C03632=1078.850,415.246,-107.346,176.673,31.266,155.541
C03633=1078.842,414.999,-107.303,176.669,31.256,155.538
C03634=1078.836,414.753,-107.261,176.663,31.246,155.536
C03635=1078.829,414.506,-107.218,176.659,31.236,155.534
C03636=1078.821,414.260,-107.176,176.654,31.226,155.532
C03637=1078.814,414.014,-107.134,176.649,31.216,155.530
C03638=1078.807,413.768,-107.091,176.645,31.206,155.528
C03639=1078.800,413.524,-107.050,176.640,31.197,155.526
C03640=1078.793,413.280,-107.008,176.635,31.187,155.523
C03641=1078.786,413.038,-106.966,176.630,31.177,155.521
C03642=1078.779,412.794,-106.924,176.626,31.167,155.519
C03643=1078.772,412.551,-106.883,176.622,31.158,155.517
C03644=1078.765,412.307,-106.841,176.617,31.148,155.515
C03645=1078.758,412.064,-106.799,176.612,31.139,155.513
C03646=1078.751,411.820,-106.757,176.607,31.129,155.511
C03647=1078.744,411.574,-106.716,176.603,31.119,155.509
C03648=1078.737,411.328,-106.674,176.599,31.110,155.507
C03649=1078.730,411.081,-106.631,176.593,31.100,155.505
C03650=1078.723,410.835,-106.590,176.589,31.091,155.503
C03651=1078.716,410.588,-106.547,176.584,31.081,155.501
C03652=1078.710,410.342,-106.506,176.580,31.072,155.499
C03653=1078.702,410.096,-106.464,176.576,31.062,155.496
C03654=1078.696,409.849,-106.422,176.570,31.053,155.494
C03655=1078.689,409.603,-106.380,176.566,31.043,155.492
C03656=1078.682,409.356,-106.338,176.562,31.034,155.490
C03657=1078.674,409.111,-106.296,176.557,31.024,155.488
C03658=1078.668,408.864,-106.255,176.553,31.015,155.486
C03659=1078.661,408.617,-106.213,176.548,31.006,155.484
C03660=1078.654,408.371,-106.171,176.543,30.996,155.482
C03661=1078.648,408.125,-106.129,176.539,30.987,155.480
C03662=1078.641,407.878,-106.088,176.534,30.977,155.478
C03663=1078.634,407.631,-106.046,176.530,30.968,155.476
C03664=1078.627,407.386,-106.005,176.526,30.959,155.474
C03665=1078.620,407.139,-105.963,176.521,30.950,155.472
C03666=1078.613,406.892,-105.922,176.517,30.941,155.470
C03667=1078.606,406.646,-105.880,176.513,30.932,155.469
C03668=1078.600,406.399,-105.839,176.508,30.922,155.466
C03669=1078.593,406.153,-105.798,176.504,30.913,155.465
C03670=1078.585,405.906,-105.757,176.500,30.904,155.463
C03671=1078.579,405.660,-105.715,176.494,30.895,155.461
C03672=1078.572,405.413,-105.674,176.490,30.886,155.459
C03673=1078.566,405.167,-105.632,176.485,30.877,155.457
C03674=1078.559,404.921,-105.591,176.481,30.869,155.455
C03675=1078.552,404.674,-105.550,176.477,30.860,155.453
C03676=1078.544,404.427,-105.509,176.472,30.851,155.451
C03677=1078.538,404.181,-105.467,176.468,30.841,155.449
C03678=1078.531,403.935,-105.426,176.464,30.833,155.448
C03679=1078.524,403.687,-105.386,176.459,30.824,155.446
C03680=1078.517,403.442,-105.345,176.455,30.815,155.444
C03681=1078.510,403.195,-105.303,176.451,30.806,155.442
C03682=1078.503,402.949,-105.263,176.446,30.798,155.440
C03683=1078.497,402.702,-105.221,176.442,30.789,155.438
C03684=1078.490,402.455,-105.180,176.438,30.780,155.436
C03685=1078.483,402.209,-105.139,176.433,30.772,155.435
C03686=1078.476,401.962,-105.099,176.429,30.763,155.433
C03687=1078.470,401.716,-105.058,176.425,30.755,155.431
C03688=1078.462,401.469,-105.017,176.421,30.746,155.429
C03689=1078.456,401.223,-104.977,176.417,30.738,155.427
C03690=1078.449,400.976,-104.935,176.413,30.729,155.426
C03691=1078.442,400.730,-104.895,176.408,30.721,155.424
C03692=1078.435,400.483,-104.854,176.404,30.712,155.422
C03693=1078.429,400.237,-104.814,176.400,30.703,155.420
C03694=1078.422,399.989,-104.773,176.395,30.695,155.418
C03695=1078.415,399.747,-104.733,176.391,30.686,155.417
C03696=1078.408,399.505,-104.693,176.387,30.678,155.415
C03697=1078.402,399.263,-104.653,176.383,30.670,155.413
C03698=1078.395,399.021,-104.613,176.379,30.662,155.411
C03699=1078.389,398.779,-104.574,176.375,30.653,155.410
C03700=1078.383,398.536,-104.535,176.370,30.645,155.408
C03701=1078.376,398.295,-104.495,176.366,30.637,155.406
C03702=1078.370,398.052,-104.455,176.363,30.629,155.405
C03703=1078.362,397.805,-104.415,176.358,30.621,155.403
C03704=1078.355,397.559,-104.374,176.354,30.613,155.401
C03705=1078.348,397.312,-104.333,176.350,30.604,155.400
C03706=1078.342,397.065,-104.293,176.345,30.596,155.398
C03707=1078.336,396.819,-104.253,176.342,30.588,155.396
C03708=1078.329,396.572,-104.213,176.338,30.580,155.394
C03709=1078.321,396.325,-104.173,176.333,30.572,155.393
C03710=1078.315,396.079,-104.133,176.329,30.564,155.391
C03711=1078.309,395.832,-104.093,176.325,30.555,155.389
C03712=1078.302,395.586,-104.053,176.320,30.547,155.388
C03713=1078.295,395.338,-104.012,176.317,30.539,155.386
C03714=1078.288,395.092,-103.973,176.313,30.531,155.384
C03715=1078.282,394.846,-103.932,176.309,30.523,155.383
C03716=1078.275,394.599,-103.892,176.304,30.515,155.381
C03717=1078.269,394.352,-103.852,176.301,30.507,155.379
C03718=1078.261,394.106,-103.812,176.297,30.499,155.378
C03719=1078.255,393.859,-103.773,176.292,30.491,155.376
C03720=1078.249,393.612,-103.733,176.288,30.484,155.375
C03721=1078.242,393.366,-103.693,176.284,30.476,155.373
C03722=1078.235,393.119,-103.653,176.280,30.468,155.371
C03723=1078.225,392.731,-103.591,176.273,30.455,155.369
C03724=1078.214,392.342,-103.528,176.268,30.443,155.366
C03725=1078.204,391.954,-103.466,176.261,30.430,155.364
C03726=1078.193,391.566,-103.403,176.255,30.418,155.361
C03727=1078.187,391.319,-103.363,176.250,30.411,155.360
C03728=1078.180,391.072,-103.324,176.246,30.403,155.358
C03729=1078.174,390.825,-103.284,176.243,30.396,155.356
C03730=1078.167,390.579,-103.245,176.238,30.388,155.355
C03731=1078.160,390.332,-103.206,176.234,30.380,155.353
C03732=1078.153,390.086,-103.166,176.230,30.372,155.352
C03733=1078.147,389.839,-103.127,176.227,30.365,155.350
C03734=1078.140,389.592,-103.087,176.222,30.357,155.349
C03735=1078.133,389.346,-103.048,176.218,30.350,155.347
C03736=1078.127,389.099,-103.009,176.215,30.343,155.346
C03737=1078.120,388.852,-102.969,176.210,30.335,155.344
C03738=1078.113,388.605,-102.930,176.206,30.327,155.343
C03739=1078.107,388.359,-102.891,176.203,30.320,155.341
C03740=1078.101,388.111,-102.852,176.198,30.312,155.340
C03741=1078.093,387.865,-102.812,176.194,30.305,155.338
C03742=1078.087,387.618,-102.774,176.191,30.298,155.337
C03743=1078.081,387.371,-102.734,176.187,30.290,155.335
C03744=1078.074,387.124,-102.695,176.182,30.283,155.334
C03745=1078.067,386.878,-102.657,176.179,30.276,155.332
C03746=1078.061,386.631,-102.616,176.175,30.268,155.331
C03747=1078.054,386.384,-102.578,176.170,30.261,155.329
C03748=1078.047,386.137,-102.539,176.167,30.253,155.328
C03749=1078.041,385.891,-102.500,176.163,30.246,155.326
C03750=1078.035,385.644,-102.461,176.159,30.239,155.325
C03751=1078.026,385.316,-102.409,176.153,30.229,155.323
C03752=1078.017,384.987,-102.357,176.148,30.219,155.321
C03753=1078.009,384.660,-102.306,176.143,30.210,155.319
C03754=1078.000,384.331,-102.254,176.138,30.200,155.317
C03755=1077.993,384.085,-102.215,176.135,30.193,155.316
C03756=1077.986,383.838,-102.176,176.131,30.186,155.314
C03757=1077.980,383.592,-102.138,176.126,30.179,155.313
C03758=1077.974,383.344,-102.099,176.123,30.171,155.311
C03759=1077.968,383.097,-102.060,176.119,30.164,155.310
C03760=1077.961,382.850,-102.021,176.115,30.157,155.308
C03761=1077.955,382.604,-101.983,176.111,30.150,155.307
C03762=1077.948,382.357,-101.945,176.108,30.143,155.306
C03763=1077.942,382.110,-101.905,176.104,30.136,155.304
C03764=1077.936,381.863,-101.867,176.099,30.129,155.303
C03765=1077.929,381.616,-101.829,176.096,30.122,155.301
C03766=1077.922,381.369,-101.790,176.092,30.114,155.300
C03767=1077.916,381.122,-101.751,176.088,30.108,155.299
C03768=1077.910,380.876,-101.713,176.084,30.101,155.297
C03769=1077.902,380.629,-101.675,176.081,30.094,155.296
C03770=1077.896,380.382,-101.637,176.077,30.087,155.294
C03771=1077.889,380.135,-101.598,176.073,30.080,155.293
C03772=1077.883,379.888,-101.560,176.069,30.073,155.292
C03773=1077.876,379.641,-101.521,176.066,30.066,155.290
C03774=1077.870,379.394,-101.483,176.061,30.059,155.289
C03775=1077.863,379.148,-101.445,176.058,30.052,155.288
C03776=1077.857,378.900,-101.407,176.054,30.046,155.286
C03777=1077.851,378.654,-101.368,176.050,30.039,155.285
C03778=1077.844,378.407,-101.330,176.046,30.032,155.284
C03779=1077.838,378.159,-101.292,176.043,30.025,155.282
C03780=1077.831,377.913,-101.254,176.039,30.018,155.281
C03781=1077.824,377.666,-101.216,176.035,30.012,155.280
C03782=1077.818,377.419,-101.178,176.031,30.005,155.278
C03783=1077.812,377.172,-101.140,176.028,29.998,155.277
C03784=1077.805,376.925,-101.101,176.023,29.991,155.276
C03785=1077.799,376.678,-101.064,176.020,29.985,155.274
C03786=1077.793,376.431,-101.025,176.016,29.978,155.273
C03787=1077.786,376.184,-100.988,176.013,29.971,155.272
C03788=1077.779,375.937,-100.950,176.009,29.965,155.270
C03789=1077.774,375.690,-100.912,176.005,29.958,155.269
C03790=1077.767,375.443,-100.874,176.002,29.951,155.268
C03791=1077.761,375.197,-100.836,175.997,29.944,155.266
C03792=1077.754,374.949,-100.798,175.994,29.938,155.265
C03793=1077.748,374.703,-100.760,175.990,29.931,155.264
C03794=1077.741,374.455,-100.722,175.987,29.925,155.263
C03795=1077.735,374.209,-100.685,175.983,29.918,155.261
C03796=1077.729,373.961,-100.646,175.979,29.911,155.260
C03797=1077.723,373.714,-100.609,175.976,29.905,155.259
C03798=1077.716,373.468,-100.572,175.971,29.898,155.257
C03799=1077.710,373.220,-100.533,175.968,29.892,155.256
C03800=1077.703,372.973,-100.497,175.965,29.886,155.255
C03801=1077.697,372.726,-100.459,175.960,29.879,155.254
C03802=1077.691,372.479,-100.421,175.957,29.872,155.252
C03803=1077.685,372.258,-100.388,175.954,29.867,155.251
C03804=1077.679,372.038,-100.354,175.950,29.861,155.250
C03805=1077.673,371.818,-100.321,175.947,29.855,155.249
C03806=1077.668,371.597,-100.287,175.944,29.849,155.248
C03807=1077.661,371.377,-100.254,175.940,29.844,155.247
C03808=1077.656,371.156,-100.221,175.937,29.838,155.246
C03809=1077.651,370.935,-100.187,175.934,29.832,155.245
C03810=1077.645,370.714,-100.154,175.931,29.827,155.244
C03811=1077.638,370.468,-100.117,175.927,29.820,155.242
C03812=1077.632,370.221,-100.079,175.924,29.814,155.241
C03813=1077.625,369.973,-100.042,175.919,29.808,155.240
C03814=1077.619,369.727,-100.004,175.916,29.802,155.239
C03815=1077.612,369.479,-99.968,175.913,29.795,155.238
C03816=1077.606,369.232,-99.930,175.908,29.789,155.236
C03817=1077.600,368.986,-99.893,175.905,29.782,155.235
C03818=1077.594,368.738,-99.856,175.902,29.776,155.234
C03819=1077.587,368.491,-99.818,175.898,29.770,155.233
C03820=1077.581,368.244,-99.781,175.894,29.764,155.232
C03821=1077.575,367.997,-99.745,175.891,29.758,155.230
C03822=1077.568,367.749,-99.706,175.887,29.751,155.229
C03823=1077.562,367.502,-99.670,175.883,29.745,155.228
C03824=1077.555,367.256,-99.633,175.880,29.739,155.227
C03825=1077.550,367.008,-99.596,175.877,29.733,155.226
C03826=1077.543,366.761,-99.559,175.873,29.726,155.224
C03827=1077.537,366.514,-99.521,175.869,29.720,155.223
C03828=1077.531,366.267,-99.485,175.866,29.714,155.222
C03829=1077.525,366.020,-99.448,175.862,29.708,155.221
C03830=1077.518,365.773,-99.411,175.858,29.702,155.220
C03831=1077.512,365.525,-99.374,175.855,29.696,155.219
C03832=1077.506,365.278,-99.337,175.851,29.689,155.217
C03833=1077.500,365.031,-99.300,175.848,29.683,155.216
C03834=1077.493,364.784,-99.264,175.844,29.677,155.215
C03835=1077.487,364.537,-99.226,175.841,29.671,155.214
C03836=1077.480,364.289,-99.189,175.837,29.666,155.213
C03837=1077.474,364.042,-99.153,175.833,29.659,155.212
C03838=1077.468,363.795,-99.116,175.830,29.653,155.211
C03839=1077.461,363.548,-99.080,175.827,29.647,155.209
C03840=1077.456,363.301,-99.043,175.822,29.641,155.208
C03841=1077.449,363.053,-99.006,175.819,29.636,155.207
C03842=1077.443,362.806,-98.970,175.816,29.630,155.206
C03843=1077.436,362.559,-98.933,175.813,29.624,155.205
C03844=1077.430,362.312,-98.897,175.808,29.617,155.204
C03845=1077.423,362.065,-98.860,175.805,29.612,155.203
C03846=1077.417,361.818,-98.824,175.802,29.606,155.202
C03847=1077.412,361.570,-98.787,175.798,29.600,155.201
C03848=1077.405,361.323,-98.750,175.794,29.594,155.199
C03849=1077.398,361.076,-98.714,175.791,29.588,155.198
C03850=1077.392,360.828,-98.678,175.787,29.582,155.197
C03851=1077.386,360.581,-98.641,175.784,29.576,155.196
C03852=1077.380,360.334,-98.605,175.781,29.571,155.195
C03853=1077.373,360.087,-98.569,175.777,29.564,155.194
C03854=1077.367,359.840,-98.532,175.773,29.559,155.193
C03855=1077.361,359.592,-98.496,175.770,29.553,155.192
C03856=1077.355,359.345,-98.460,175.767,29.547,155.191
C03857=1077.348,359.098,-98.423,175.763,29.541,155.190
C03858=1077.342,358.851,-98.387,175.759,29.535,155.188
C03859=1077.337,358.638,-98.356,175.757,29.531,155.188
C03860=1077.331,358.426,-98.325,175.753,29.526,155.187
C03861=1077.326,358.213,-98.294,175.750,29.521,155.186
C03862=1077.320,358.001,-98.263,175.747,29.516,155.185
C03863=1077.315,357.789,-98.232,175.744,29.511,155.184
C03864=1077.309,357.576,-98.201,175.742,29.506,155.183
C03865=1077.305,357.364,-98.170,175.738,29.501,155.182
C03866=1077.299,357.152,-98.139,175.736,29.496,155.181
C03867=1077.293,356.905,-98.103,175.732,29.490,155.180
C03868=1077.287,356.657,-98.067,175.728,29.485,155.179
C03869=1077.280,356.410,-98.031,175.725,29.479,155.178
C03870=1077.274,356.162,-97.995,175.722,29.474,155.177
C03871=1077.268,355.915,-97.959,175.718,29.468,155.176
C03872=1077.262,355.667,-97.923,175.715,29.462,155.175
C03873=1077.255,355.420,-97.887,175.711,29.456,155.174
C03874=1077.249,355.173,-97.851,175.707,29.451,155.173
C03875=1077.243,354.925,-97.816,175.704,29.445,155.172
C03876=1077.236,354.678,-97.779,175.701,29.439,155.171
C03877=1077.231,354.431,-97.744,175.698,29.434,155.170
C03878=1077.225,354.184,-97.708,175.694,29.428,155.169
C03879=1077.219,353.937,-97.672,175.691,29.423,155.168
C03880=1077.212,353.689,-97.636,175.688,29.417,155.167
C03881=1077.206,353.442,-97.601,175.683,29.411,155.166
C03882=1077.200,353.194,-97.565,175.680,29.406,155.165
C03883=1077.193,352.947,-97.529,175.677,29.400,155.164
C03884=1077.188,352.700,-97.493,175.673,29.395,155.163
C03885=1077.181,352.452,-97.458,175.670,29.390,155.162
C03886=1077.175,352.205,-97.422,175.667,29.384,155.161
C03887=1077.169,351.957,-97.387,175.664,29.378,155.160
C03888=1077.162,351.710,-97.352,175.660,29.373,155.159
C03889=1077.156,351.463,-97.315,175.657,29.368,155.158
C03890=1077.150,351.215,-97.279,175.653,29.362,155.157
C03891=1077.144,350.968,-97.245,175.649,29.356,155.156
C03892=1077.138,350.721,-97.209,175.646,29.351,155.155
C03893=1077.132,350.473,-97.173,175.643,29.346,155.154
C03894=1077.125,350.226,-97.138,175.639,29.340,155.153
C03895=1077.119,349.978,-97.102,175.636,29.335,155.152
C03896=1077.113,349.731,-97.068,175.633,29.330,155.151
C03897=1077.107,349.484,-97.032,175.629,29.324,155.150
C03898=1077.100,349.236,-96.997,175.626,29.319,155.149
C03899=1077.094,348.988,-96.962,175.623,29.313,155.148
C03900=1077.089,348.741,-96.926,175.620,29.308,155.147
C03901=1077.082,348.494,-96.891,175.616,29.303,155.146
C03902=1077.076,348.246,-96.855,175.613,29.297,155.145
C03903=1077.069,347.999,-96.820,175.610,29.292,155.144
C03904=1077.064,347.752,-96.785,175.605,29.286,155.143
C03905=1077.057,347.504,-96.750,175.602,29.281,155.142
C03906=1077.051,347.256,-96.715,175.599,29.275,155.141
C03907=1077.045,347.009,-96.680,175.595,29.270,155.140
C03908=1077.039,346.762,-96.644,175.592,29.265,155.139
C03909=1077.033,346.514,-96.610,175.589,29.260,155.138
C03910=1077.027,346.267,-96.574,175.585,29.255,155.137
C03911=1077.020,346.019,-96.539,175.582,29.249,155.136
C03912=1077.014,345.772,-96.504,175.579,29.244,155.135
C03913=1077.009,345.524,-96.470,175.576,29.239,155.134
C03914=1077.003,345.277,-96.434,175.572,29.233,155.133
C03915=1076.997,345.066,-96.404,175.570,29.229,155.133
C03916=1076.992,344.855,-96.375,175.566,29.224,155.132
C03917=1076.987,344.645,-96.345,175.564,29.220,155.131
C03918=1076.982,344.434,-96.316,175.562,29.216,155.130
C03919=1076.977,344.223,-96.285,175.558,29.211,155.129
C03920=1076.971,344.013,-96.255,175.556,29.207,155.129
C03921=1076.966,343.802,-96.226,175.552,29.202,155.128
C03922=1076.960,343.591,-96.197,175.550,29.198,155.127
C03923=1076.955,343.343,-96.162,175.547,29.193,155.126
C03924=1076.948,343.096,-96.127,175.543,29.188,155.125
C03925=1076.942,342.848,-96.092,175.540,29.183,155.124
C03926=1076.935,342.601,-96.057,175.537,29.177,155.123
C03927=1076.930,342.353,-96.023,175.533,29.172,155.122
C03928=1076.924,342.105,-95.988,175.530,29.167,155.121
C03929=1076.917,341.859,-95.954,175.527,29.162,155.121
C03930=1076.911,341.611,-95.919,175.523,29.156,155.120
C03931=1076.906,341.363,-95.884,175.520,29.151,155.119
C03932=1076.899,341.116,-95.849,175.517,29.146,155.118
C03933=1076.893,340.868,-95.815,175.514,29.141,155.117
C03934=1076.887,340.620,-95.781,175.510,29.136,155.116
C03935=1076.881,340.374,-95.746,175.507,29.131,155.115
C03936=1076.875,340.125,-95.711,175.504,29.126,155.114
C03937=1076.869,339.878,-95.677,175.500,29.121,155.113
C03938=1076.862,339.630,-95.643,175.497,29.116,155.112
C03939=1076.856,339.383,-95.608,175.494,29.111,155.112
C03940=1076.850,339.135,-95.573,175.491,29.106,155.111
C03941=1076.844,338.888,-95.539,175.488,29.101,155.110
C03942=1076.838,338.640,-95.504,175.485,29.095,155.109
C03943=1076.832,338.393,-95.470,175.481,29.091,155.108
C03944=1076.826,338.145,-95.436,175.478,29.086,155.107
C03945=1076.820,337.897,-95.402,175.475,29.081,155.106
C03946=1076.814,337.649,-95.367,175.471,29.076,155.105
C03947=1076.808,337.402,-95.333,175.468,29.070,155.104
C03948=1076.801,337.154,-95.299,175.465,29.066,155.104
C03949=1076.795,336.907,-95.265,175.461,29.061,155.103
C03950=1076.790,336.660,-95.231,175.458,29.056,155.102
C03951=1076.783,336.412,-95.196,175.455,29.050,155.101
C03952=1076.777,336.164,-95.162,175.452,29.046,155.100
C03953=1076.771,335.916,-95.128,175.449,29.041,155.099
C03954=1076.765,335.669,-95.094,175.446,29.036,155.098
C03955=1076.758,335.421,-95.059,175.443,29.031,155.098
C03956=1076.753,335.174,-95.025,175.439,29.026,155.097
C03957=1076.747,334.926,-94.991,175.436,29.021,155.096
C03958=1076.740,334.678,-94.957,175.433,29.016,155.095
C03959=1076.735,334.431,-94.924,175.429,29.011,155.094
C03960=1076.729,334.183,-94.890,175.426,29.006,155.093
C03961=1076.722,333.936,-94.856,175.424,29.002,155.092
C03962=1076.716,333.688,-94.822,175.420,28.997,155.092
C03963=1076.710,333.441,-94.788,175.417,28.992,155.091
C03964=1076.704,333.192,-94.754,175.414,28.987,155.090
C03965=1076.698,332.945,-94.720,175.410,28.982,155.089
C03966=1076.692,332.698,-94.686,175.407,28.977,155.088
C03967=1076.686,332.449,-94.652,175.404,28.972,155.087
C03968=1076.680,332.202,-94.618,175.400,28.967,155.087
C03969=1076.674,331.955,-94.584,175.398,28.962,155.086
C03970=1076.669,331.707,-94.551,175.395,28.958,155.085
C03971=1076.662,331.494,-94.522,175.391,28.953,155.084
C03972=1076.657,331.280,-94.492,175.389,28.949,155.083
C03973=1076.653,331.067,-94.463,175.387,28.946,155.083
C03974=1076.647,330.853,-94.435,175.384,28.941,155.082
C03975=1076.641,330.640,-94.405,175.381,28.937,155.081
C03976=1076.636,330.426,-94.376,175.378,28.933,155.081
C03977=1076.631,330.214,-94.348,175.376,28.929,155.080
C03978=1076.625,330.000,-94.319,175.372,28.925,155.079
C03979=1076.620,329.752,-94.285,175.369,28.920,155.078
C03980=1076.613,329.504,-94.252,175.367,28.916,155.078
C03981=1076.607,329.257,-94.218,175.363,28.911,155.077
C03982=1076.600,329.009,-94.185,175.360,28.906,155.076
C03983=1076.595,328.761,-94.151,175.357,28.901,155.075
C03984=1076.588,328.514,-94.118,175.353,28.897,155.074
C03985=1076.582,328.266,-94.084,175.351,28.892,155.074
C03986=1076.576,328.019,-94.051,175.348,28.888,155.073
C03987=1076.570,327.771,-94.017,175.344,28.883,155.072
C03988=1076.563,327.523,-93.984,175.341,28.878,155.071
C03989=1076.557,327.275,-93.950,175.338,28.873,155.070
C03990=1076.551,327.028,-93.918,175.334,28.869,155.070
C03991=1076.545,326.780,-93.884,175.332,28.864,155.069
C03992=1076.539,326.532,-93.851,175.329,28.860,155.068
C03993=1076.533,326.284,-93.817,175.325,28.854,155.067
C03994=1076.527,326.036,-93.784,175.322,28.850,155.066
C03995=1076.521,325.789,-93.751,175.320,28.845,155.066
C03996=1076.515,325.541,-93.718,175.316,28.841,155.065
C03997=1076.509,325.294,-93.684,175.313,28.836,155.064
C03998=1076.502,325.046,-93.651,175.310,28.832,155.063
C03999=1076.497,324.798,-93.618,175.306,28.827,155.063
C04000=1076.490,324.550,-93.585,175.304,28.822,155.062
C04001=1076.484,324.302,-93.552,175.301,28.818,155.061
C04002=1076.478,324.054,-93.519,175.298,28.813,155.060
C04003=1076.473,323.807,-93.486,175.294,28.808,155.059
C04004=1076.466,323.559,-93.453,175.292,28.804,155.059
C04005=1076.460,323.312,-93.419,175.289,28.799,155.058
C04006=1076.454,323.064,-93.386,175.285,28.794,155.057
C04007=1076.449,322.816,-93.353,175.282,28.790,155.056
C04008=1076.442,322.569,-93.320,175.280,28.785,155.055
C04009=1076.436,322.321,-93.287,175.276,28.781,155.055
C04010=1076.430,322.073,-93.254,175.273,28.776,155.054
C04011=1076.424,321.826,-93.221,175.270,28.771,155.053
C04012=1076.419,321.577,-93.189,175.267,28.767,155.052
C04013=1076.413,321.329,-93.156,175.264,28.762,155.052
C04014=1076.406,321.082,-93.123,175.261,28.758,155.051
C04015=1076.401,320.834,-93.090,175.258,28.753,155.050
C04016=1076.394,320.586,-93.057,175.255,28.749,155.049
C04017=1076.389,320.338,-93.024,175.252,28.744,155.048
C04018=1076.383,320.091,-92.991,175.248,28.739,155.048
C04019=1076.376,319.843,-92.958,175.246,28.735,155.047
C04020=1076.371,319.595,-92.925,175.243,28.730,155.046
C04021=1076.365,319.347,-92.893,175.239,28.726,155.045
C04022=1076.358,319.100,-92.860,175.237,28.721,155.045
C04023=1076.353,318.852,-92.827,175.234,28.717,155.044
C04024=1076.347,318.604,-92.794,175.230,28.712,155.043
C04025=1076.341,318.357,-92.762,175.227,28.708,155.042
C04026=1076.336,318.109,-92.729,175.225,28.703,155.042
C04027=1076.330,317.892,-92.701,175.222,28.699,155.041
C04028=1076.325,317.675,-92.672,175.219,28.695,155.040
C04029=1076.321,317.459,-92.643,175.216,28.691,155.040
C04030=1076.315,317.242,-92.615,175.214,28.687,155.039
C04031=1076.310,317.026,-92.586,175.212,28.683,155.038
C04032=1076.304,316.809,-92.557,175.208,28.679,155.038
C04033=1076.300,316.593,-92.529,175.206,28.675,155.037
C04034=1076.294,316.376,-92.501,175.203,28.671,155.036
C04035=1076.289,316.127,-92.468,175.200,28.666,155.035
C04036=1076.282,315.880,-92.435,175.198,28.663,155.035
C04037=1076.277,315.632,-92.404,175.194,28.658,155.034
C04038=1076.271,315.384,-92.370,175.191,28.653,155.033
C04039=1076.265,315.137,-92.337,175.189,28.649,155.032
C04040=1076.259,314.889,-92.305,175.185,28.644,155.032
C04041=1076.253,314.642,-92.273,175.182,28.640,155.031
C04042=1076.247,314.393,-92.241,175.180,28.636,155.030
C04043=1076.241,314.145,-92.209,175.176,28.631,155.030
C04044=1076.235,313.898,-92.176,175.173,28.627,155.029
C04045=1076.229,313.649,-92.144,175.171,28.622,155.028
C04046=1076.223,313.402,-92.112,175.167,28.618,155.027
C04047=1076.217,313.154,-92.079,175.164,28.614,155.027
C04048=1076.210,312.906,-92.048,175.162,28.610,155.026
C04049=1076.204,312.659,-92.016,175.158,28.605,155.025
C04050=1076.198,312.411,-91.984,175.155,28.601,155.025
C04051=1076.192,312.162,-91.952,175.153,28.596,155.024
C04052=1076.186,311.915,-91.919,175.149,28.592,155.023
C04053=1076.180,311.667,-91.887,175.146,28.588,155.022
C04054=1076.174,311.419,-91.856,175.144,28.584,155.022
C04055=1076.168,311.172,-91.823,175.140,28.579,155.021
C04056=1076.162,310.924,-91.791,175.138,28.575,155.020
C04057=1076.156,310.675,-91.759,175.135,28.570,155.020
C04058=1076.150,310.428,-91.727,175.131,28.566,155.019
C04059=1076.144,310.180,-91.696,175.129,28.562,155.018
C04060=1076.137,309.932,-91.663,175.126,28.558,155.017
C04061=1076.131,309.684,-91.631,175.122,28.553,155.017
C04062=1076.126,309.437,-91.599,175.120,28.549,155.016
C04063=1076.120,309.188,-91.567,175.117,28.544,155.015
C04064=1076.113,308.941,-91.536,175.113,28.540,155.015
C04065=1076.107,308.692,-91.504,175.111,28.536,155.014
C04066=1076.102,308.445,-91.472,175.108,28.532,155.013
C04067=1076.096,308.197,-91.440,175.105,28.528,155.013
C04068=1076.089,307.949,-91.408,175.102,28.523,155.012
C04069=1076.084,307.702,-91.376,175.099,28.519,155.011
C04070=1076.078,307.454,-91.344,175.096,28.514,155.010
C04071=1076.072,307.206,-91.313,175.093,28.510,155.010
C04072=1076.065,306.958,-91.281,175.091,28.506,155.009
C04073=1076.059,306.710,-91.249,175.087,28.502,155.008
C04074=1076.054,306.462,-91.218,175.084,28.497,155.008
C04075=1076.047,306.215,-91.186,175.082,28.493,155.007
C04076=1076.041,305.966,-91.154,175.078,28.489,155.006
C04077=1076.036,305.719,-91.123,175.076,28.485,155.006
C04078=1076.030,305.471,-91.091,175.073,28.480,155.005
C04079=1076.024,305.223,-91.060,175.069,28.476,155.004
C04080=1076.018,304.975,-91.028,175.067,28.472,155.003
C04081=1076.013,304.727,-90.996,175.064,28.467,155.003
C04082=1076.006,304.479,-90.965,175.061,28.463,155.002
C04083=1076.002,304.264,-90.938,175.059,28.460,155.001
C04084=1075.996,304.049,-90.911,175.055,28.456,155.001
C04085=1075.992,303.834,-90.882,175.053,28.452,155.000
C04086=1075.986,303.619,-90.855,175.051,28.449,155.000
C04087=1075.980,303.404,-90.828,175.048,28.445,154.999
C04088=1075.976,303.189,-90.801,175.046,28.441,154.998
C04089=1075.971,302.974,-90.774,175.043,28.437,154.998
C04090=1075.965,302.759,-90.746,175.041,28.433,154.997
C04091=1075.960,302.511,-90.715,175.038,28.429,154.997
C04092=1075.954,302.263,-90.683,175.035,28.425,154.996
C04093=1075.948,302.016,-90.652,175.032,28.421,154.995
C04094=1075.942,301.767,-90.620,175.030,28.417,154.994
C04095=1075.936,301.520,-90.590,175.026,28.412,154.994
C04096=1075.931,301.272,-90.558,175.024,28.408,154.993
C04097=1075.925,301.024,-90.526,175.021,28.404,154.992
C04098=1075.919,300.776,-90.496,175.018,28.400,154.992
C04099=1075.913,300.528,-90.464,175.015,28.395,154.991
C04100=1075.908,300.280,-90.433,175.012,28.391,154.990
C04101=1075.901,300.032,-90.401,175.009,28.387,154.990
C04102=1075.896,299.784,-90.370,175.006,28.382,154.989
C04103=1075.890,299.537,-90.339,175.004,28.378,154.988
C04104=1075.884,299.288,-90.307,175.000,28.374,154.988
C04105=1075.878,299.041,-90.277,174.998,28.370,154.987
C04106=1075.873,298.793,-90.245,174.995,28.366,154.986
C04107=1075.867,298.544,-90.214,174.992,28.362,154.986
C04108=1075.861,298.297,-90.183,174.989,28.357,154.985
C04109=1075.856,298.049,-90.152,174.987,28.353,154.984
C04110=1075.849,297.801,-90.120,174.983,28.349,154.984
C04111=1075.844,297.553,-90.090,174.981,28.345,154.983
C04112=1075.838,297.304,-90.059,174.978,28.340,154.982
C04113=1075.832,297.057,-90.028,174.975,28.336,154.981
C04114=1075.826,296.809,-89.997,174.972,28.332,154.981
C04115=1075.820,296.560,-89.966,174.970,28.328,154.980
C04116=1075.814,296.313,-89.935,174.966,28.324,154.980
C04117=1075.808,296.064,-89.904,174.964,28.320,154.979
C04118=1075.802,295.817,-89.873,174.961,28.316,154.978
C04119=1075.796,295.569,-89.842,174.958,28.311,154.977
C04120=1075.791,295.321,-89.811,174.955,28.307,154.977
C04121=1075.785,295.073,-89.781,174.953,28.303,154.976
C04122=1075.779,294.825,-89.750,174.949,28.299,154.976
C04123=1075.772,294.577,-89.719,174.947,28.295,154.975
C04124=1075.766,294.329,-89.688,174.944,28.291,154.974
C04125=1075.761,294.081,-89.658,174.941,28.287,154.974
C04126=1075.755,293.833,-89.627,174.938,28.283,154.973
C04127=1075.749,293.585,-89.596,174.936,28.279,154.972
C04128=1075.743,293.337,-89.565,174.932,28.274,154.972
C04129=1075.737,293.089,-89.535,174.930,28.270,154.971
C04130=1075.731,292.841,-89.504,174.927,28.266,154.970
C04131=1075.726,292.593,-89.473,174.924,28.262,154.970
C04132=1075.720,292.345,-89.443,174.921,28.258,154.969
C04133=1075.713,292.097,-89.412,174.919,28.254,154.968
C04134=1075.708,291.849,-89.382,174.916,28.250,154.968
C04135=1075.702,291.601,-89.352,174.913,28.246,154.967
C04136=1075.696,291.352,-89.320,174.910,28.242,154.966
C04137=1075.690,291.104,-89.290,174.907,28.238,154.966
C04138=1075.684,290.857,-89.260,174.905,28.234,154.965
C04139=1075.675,290.441,-89.209,174.900,28.227,154.964
C04140=1075.664,290.026,-89.157,174.895,28.220,154.963
C04141=1075.655,289.610,-89.106,174.890,28.213,154.962
C04142=1075.645,289.195,-89.056,174.886,28.206,154.961
C04143=1075.640,288.947,-89.026,174.883,28.202,154.960
C04144=1075.633,288.698,-88.995,174.881,28.199,154.960
C04145=1075.627,288.450,-88.964,174.877,28.194,154.959
C04146=1075.621,288.203,-88.934,174.875,28.190,154.958
C04147=1075.615,287.955,-88.904,174.873,28.186,154.958
C04148=1075.609,287.706,-88.874,174.869,28.182,154.957
C04149=1075.603,287.458,-88.844,174.867,28.178,154.956
C04150=1075.597,287.210,-88.814,174.864,28.174,154.956
C04151=1075.591,286.963,-88.783,174.861,28.170,154.955
C04152=1075.586,286.714,-88.754,174.858,28.166,154.955
C04153=1075.579,286.466,-88.723,174.856,28.162,154.954
C04154=1075.574,286.218,-88.693,174.853,28.158,154.953
C04155=1075.568,285.970,-88.662,174.850,28.154,154.953
C04156=1075.562,285.722,-88.633,174.848,28.150,154.952
C04157=1075.556,285.474,-88.603,174.844,28.146,154.951
C04158=1075.550,285.226,-88.572,174.842,28.142,154.951
C04159=1075.544,284.978,-88.543,174.840,28.138,154.950
C04160=1075.538,284.729,-88.512,174.836,28.134,154.949
C04161=1075.532,284.481,-88.482,174.834,28.130,154.949
C04162=1075.527,284.233,-88.452,174.831,28.126,154.948
C04163=1075.521,283.985,-88.422,174.828,28.122,154.948
C04164=1075.515,283.737,-88.393,174.826,28.118,154.947
C04165=1075.509,283.489,-88.362,174.823,28.114,154.946
C04166=1075.503,283.241,-88.333,174.820,28.110,154.946
C04167=1075.497,282.993,-88.302,174.817,28.106,154.945
C04168=1075.492,282.744,-88.273,174.815,28.102,154.944
C04169=1075.486,282.497,-88.242,174.812,28.098,154.944
C04170=1075.480,282.249,-88.213,174.809,28.094,154.943
C04171=1075.474,282.001,-88.183,174.807,28.090,154.942
C04172=1075.469,281.752,-88.153,174.804,28.086,154.942
C04173=1075.463,281.504,-88.123,174.801,28.082,154.941
C04174=1075.457,281.256,-88.093,174.799,28.078,154.941
C04175=1075.451,281.007,-88.063,174.795,28.074,154.940
C04176=1075.445,280.759,-88.034,174.793,28.070,154.939
C04177=1075.439,280.511,-88.004,174.791,28.066,154.939
C04178=1075.433,280.263,-87.974,174.787,28.062,154.938
C04179=1075.427,280.015,-87.945,174.785,28.058,154.937
C04180=1075.421,279.766,-87.915,174.783,28.054,154.937
C04181=1075.415,279.519,-87.885,174.779,28.050,154.936
C04182=1075.409,279.271,-87.856,174.777,28.046,154.936
C04183=1075.404,279.022,-87.826,174.775,28.042,154.935
C04184=1075.398,278.774,-87.797,174.771,28.038,154.934
C04185=1075.392,278.526,-87.767,174.769,28.034,154.934
C04186=1075.386,278.278,-87.737,174.766,28.031,154.933
C04187=1075.380,278.030,-87.708,174.763,28.027,154.933
C04188=1075.375,277.781,-87.678,174.761,28.023,154.932
C04189=1075.368,277.534,-87.649,174.758,28.018,154.931
C04190=1075.362,277.285,-87.619,174.755,28.015,154.931
C04191=1075.353,276.880,-87.570,174.751,28.008,154.930
C04192=1075.343,276.474,-87.523,174.746,28.002,154.929
C04193=1075.334,276.069,-87.474,174.743,27.995,154.928
C04194=1075.325,275.664,-87.427,174.738,27.989,154.927
C04195=1075.319,275.416,-87.397,174.735,27.985,154.926
C04196=1075.313,275.168,-87.368,174.733,27.981,154.925
C04197=1075.307,274.919,-87.338,174.730,27.977,154.925
C04198=1075.301,274.671,-87.309,174.727,27.973,154.924
C04199=1075.295,274.423,-87.280,174.725,27.969,154.924
C04200=1075.289,274.174,-87.251,174.722,27.965,154.923
C04201=1075.284,273.926,-87.221,174.719,27.961,154.922
C04202=1075.277,273.678,-87.192,174.717,27.957,154.922
C04203=1075.272,273.429,-87.162,174.715,27.953,154.921
C04204=1075.266,273.182,-87.134,174.711,27.950,154.921
C04205=1075.260,272.933,-87.105,174.709,27.946,154.920
C04206=1075.255,272.685,-87.076,174.707,27.942,154.919
C04207=1075.249,272.437,-87.047,174.703,27.938,154.919
C04208=1075.242,272.189,-87.018,174.701,27.934,154.918
C04209=1075.237,271.940,-86.988,174.699,27.930,154.917
C04210=1075.230,271.692,-86.959,174.695,27.926,154.917
C04211=1075.224,271.444,-86.930,174.693,27.922,154.916
C04212=1075.219,271.196,-86.901,174.691,27.918,154.916
C04213=1075.213,270.947,-86.872,174.688,27.915,154.915
C04214=1075.207,270.699,-86.843,174.685,27.911,154.915
C04215=1075.202,270.451,-86.814,174.683,27.907,154.914
C04216=1075.195,270.203,-86.785,174.680,27.903,154.913
C04217=1075.189,269.954,-86.756,174.677,27.899,154.913
C04218=1075.185,269.706,-86.727,174.675,27.895,154.912
C04219=1075.178,269.458,-86.698,174.672,27.891,154.912
C04220=1075.172,269.210,-86.669,174.670,27.887,154.911
C04221=1075.166,268.961,-86.641,174.667,27.883,154.910
C04222=1075.161,268.713,-86.611,174.664,27.880,154.910
C04223=1075.155,268.465,-86.582,174.662,27.876,154.909
C04224=1075.149,268.216,-86.554,174.659,27.871,154.908
C04225=1075.143,267.968,-86.525,174.656,27.868,154.908
C04226=1075.136,267.720,-86.496,174.654,27.864,154.907
C04227=1075.132,267.472,-86.467,174.652,27.860,154.907
C04228=1075.126,267.224,-86.438,174.648,27.856,154.906
C04229=1075.120,266.975,-86.410,174.646,27.852,154.905
C04230=1075.113,266.727,-86.381,174.644,27.849,154.905
C04231=1075.108,266.479,-86.352,174.641,27.845,154.904
C04232=1075.102,266.231,-86.324,174.638,27.840,154.904
C04233=1075.096,265.982,-86.294,174.636,27.837,154.903
C04234=1075.090,265.733,-86.266,174.634,27.833,154.902
C04235=1075.085,265.486,-86.237,174.631,27.829,154.902
C04236=1075.079,265.237,-86.209,174.628,27.825,154.901
C04237=1075.073,264.989,-86.180,174.626,27.821,154.901
C04238=1075.067,264.741,-86.152,174.623,27.818,154.900
C04239=1075.061,264.492,-86.124,174.621,27.814,154.900
C04240=1075.055,264.244,-86.095,174.618,27.809,154.899
C04241=1075.050,263.995,-86.066,174.615,27.806,154.898
C04242=1075.044,263.748,-86.037,174.613,27.802,154.898
C04243=1075.034,263.345,-85.992,174.609,27.796,154.897
C04244=1075.024,262.943,-85.945,174.604,27.789,154.896
C04245=1075.015,262.541,-85.900,174.600,27.784,154.895
C04246=1075.005,262.139,-85.853,174.596,27.778,154.894
C04247=1074.999,261.890,-85.825,174.594,27.774,154.893
C04248=1074.993,261.641,-85.797,174.592,27.770,154.893
C04249=1074.987,261.393,-85.769,174.588,27.766,154.892
C04250=1074.981,261.145,-85.740,174.586,27.762,154.892
C04251=1074.975,260.897,-85.712,174.584,27.758,154.891
C04252=1074.969,260.649,-85.684,174.581,27.755,154.891
C04253=1074.963,260.400,-85.656,174.578,27.750,154.890
C04254=1074.957,260.151,-85.627,174.576,27.747,154.889
C04255=1074.952,259.904,-85.599,174.573,27.743,154.889
C04256=1074.946,259.655,-85.570,174.571,27.740,154.888
C04257=1074.939,259.407,-85.543,174.569,27.735,154.888
C04258=1074.934,259.159,-85.515,174.565,27.732,154.887
C04259=1074.928,258.910,-85.486,174.563,27.728,154.886
C04260=1074.922,258.661,-85.458,174.561,27.724,154.886
C04261=1074.916,258.413,-85.431,174.558,27.720,154.885
C04262=1074.910,258.165,-85.402,174.556,27.717,154.885
C04263=1074.904,257.917,-85.374,174.553,27.712,154.884
C04264=1074.898,257.668,-85.345,174.550,27.709,154.884
C04265=1074.892,257.420,-85.317,174.548,27.705,154.883
C04266=1074.886,257.172,-85.290,174.546,27.701,154.882
C04267=1074.880,256.923,-85.261,174.543,27.697,154.882
C04268=1074.875,256.675,-85.233,174.540,27.694,154.881
C04269=1074.869,256.426,-85.205,174.538,27.690,154.881
C04270=1074.863,256.179,-85.178,174.535,27.686,154.880
C04271=1074.857,255.930,-85.149,174.533,27.682,154.879
C04272=1074.852,255.682,-85.122,174.531,27.679,154.879
C04273=1074.846,255.432,-85.094,174.529,27.675,154.878
C04274=1074.839,255.184,-85.066,174.525,27.670,154.878
C04275=1074.834,254.936,-85.038,174.523,27.667,154.877
C04276=1074.828,254.687,-85.010,174.521,27.663,154.876
C04277=1074.822,254.439,-84.983,174.518,27.659,154.876
C04278=1074.816,254.191,-84.954,174.516,27.655,154.875
C04279=1074.811,253.943,-84.926,174.514,27.652,154.875
C04280=1074.805,253.695,-84.898,174.510,27.647,154.874
C04281=1074.799,253.446,-84.871,174.508,27.644,154.874
C04282=1074.794,253.198,-84.843,174.506,27.640,154.873
C04283=1074.788,252.949,-84.815,174.503,27.636,154.872
C04284=1074.782,252.701,-84.788,174.501,27.632,154.872
C04285=1074.776,252.452,-84.759,174.499,27.628,154.871
C04286=1074.771,252.204,-84.732,174.496,27.625,154.871
C04287=1074.764,251.955,-84.704,174.493,27.621,154.870
C04288=1074.759,251.707,-84.676,174.491,27.617,154.869
C04289=1074.753,251.459,-84.648,174.489,27.613,154.869
C04290=1074.747,251.210,-84.621,174.486,27.609,154.868
C04291=1074.741,250.962,-84.593,174.484,27.605,154.868
C04292=1074.736,250.713,-84.565,174.482,27.601,154.867
C04293=1074.730,250.465,-84.538,174.478,27.598,154.867
C04294=1074.724,250.217,-84.511,174.476,27.594,154.866
C04295=1074.715,249.811,-84.465,174.472,27.587,154.865
C04296=1074.705,249.407,-84.421,174.468,27.581,154.864
C04297=1074.696,249.002,-84.376,174.464,27.575,154.863
C04298=1074.687,248.597,-84.330,174.461,27.568,154.862
C04299=1074.681,248.349,-84.303,174.458,27.565,154.861
C04300=1074.676,248.100,-84.275,174.456,27.561,154.861
C04301=1074.670,247.852,-84.248,174.454,27.557,154.860
C04302=1074.664,247.603,-84.221,174.451,27.553,154.860
C04303=1074.658,247.355,-84.193,174.448,27.549,154.859
C04304=1074.653,247.107,-84.166,174.446,27.545,154.858
C04305=1074.647,246.859,-84.138,174.444,27.541,154.858
C04306=1074.641,246.609,-84.111,174.441,27.538,154.857
C04307=1074.636,246.361,-84.084,174.439,27.534,154.857
C04308=1074.630,246.113,-84.056,174.437,27.530,154.856
C04309=1074.624,245.864,-84.029,174.434,27.526,154.855
C04310=1074.618,245.616,-84.001,174.432,27.522,154.855
C04311=1074.612,245.368,-83.975,174.430,27.519,154.854
C04312=1074.607,245.118,-83.947,174.427,27.514,154.854
C04313=1074.601,244.871,-83.920,174.424,27.511,154.853
C04314=1074.596,244.622,-83.892,174.422,27.507,154.853
C04315=1074.589,244.373,-83.865,174.420,27.503,154.852
C04316=1074.583,244.125,-83.838,174.417,27.499,154.851
C04317=1074.578,243.876,-83.811,174.415,27.496,154.851
C04318=1074.572,243.628,-83.784,174.413,27.492,154.850
C04319=1074.566,243.380,-83.756,174.410,27.488,154.850
C04320=1074.561,243.131,-83.729,174.408,27.484,154.849
C04321=1074.555,242.883,-83.703,174.406,27.480,154.848
C04322=1074.549,242.635,-83.675,174.404,27.476,154.848
C04323=1074.543,242.385,-83.648,174.401,27.472,154.847
C04324=1074.537,242.137,-83.621,174.398,27.469,154.847
C04325=1074.532,241.889,-83.594,174.396,27.465,154.846
C04326=1074.526,241.640,-83.568,174.393,27.461,154.846
C04327=1074.519,241.392,-83.540,174.391,27.458,154.845
C04328=1074.514,241.143,-83.513,174.389,27.453,154.844
C04329=1074.508,240.895,-83.486,174.386,27.450,154.844
C04330=1074.503,240.647,-83.459,174.384,27.446,154.843
C04331=1074.496,240.397,-83.432,174.382,27.442,154.843
C04332=1074.490,240.149,-83.406,174.380,27.438,154.842
C04333=1074.485,239.901,-83.379,174.377,27.435,154.842
C04334=1074.480,239.652,-83.352,174.375,27.431,154.841
C04335=1074.473,239.403,-83.325,174.373,27.427,154.840
C04336=1074.467,239.155,-83.297,174.370,27.423,154.840
C04337=1074.461,238.907,-83.271,174.368,27.420,154.839
C04338=1074.456,238.659,-83.244,174.366,27.416,154.839
C04339=1074.450,238.410,-83.218,174.363,27.412,154.838
C04340=1074.443,238.161,-83.191,174.360,27.408,154.837
C04341=1074.438,237.913,-83.164,174.358,27.404,154.837
C04342=1074.432,237.664,-83.137,174.356,27.400,154.836
C04343=1074.426,237.416,-83.111,174.353,27.397,154.836
C04344=1074.421,237.167,-83.085,174.351,27.393,154.835
C04345=1074.416,236.918,-83.057,174.349,27.389,154.835
C04346=1074.409,236.669,-83.030,174.347,27.385,154.834
C04347=1074.400,236.259,-82.986,174.343,27.379,154.833
C04348=1074.390,235.847,-82.942,174.339,27.372,154.832
C04349=1074.381,235.435,-82.898,174.335,27.366,154.831
C04350=1074.371,235.024,-82.854,174.331,27.360,154.830
C04351=1074.365,234.775,-82.828,174.329,27.356,154.830
C04352=1074.359,234.527,-82.801,174.327,27.352,154.829
C04353=1074.354,234.278,-82.774,174.324,27.348,154.828
C04354=1074.348,234.030,-82.748,174.322,27.344,154.828
C04355=1074.342,233.782,-82.721,174.320,27.341,154.827
C04356=1074.337,233.533,-82.695,174.318,27.337,154.827
C04357=1074.331,233.284,-82.669,174.315,27.333,154.826
C04358=1074.325,233.036,-82.642,174.313,27.329,154.825
C04359=1074.319,232.788,-82.615,174.311,27.325,154.825
C04360=1074.314,232.539,-82.589,174.308,27.321,154.824
C04361=1074.308,232.290,-82.563,174.306,27.318,154.824
C04362=1074.301,232.042,-82.537,174.304,27.314,154.823
C04363=1074.296,231.793,-82.511,174.302,27.310,154.823
C04364=1074.290,231.544,-82.484,174.299,27.306,154.822
C04365=1074.284,231.296,-82.457,174.297,27.303,154.821
C04366=1074.278,231.047,-82.431,174.295,27.299,154.821
C04367=1074.273,230.798,-82.404,174.292,27.295,154.820
C04368=1074.267,230.550,-82.378,174.290,27.291,154.820
C04369=1074.261,230.301,-82.352,174.288,27.287,154.819
C04370=1074.256,230.053,-82.325,174.286,27.283,154.818
C04371=1074.249,229.804,-82.300,174.283,27.280,154.818
C04372=1074.244,229.556,-82.273,174.281,27.276,154.817
C04373=1074.238,229.307,-82.247,174.279,27.272,154.817
C04374=1074.232,229.059,-82.221,174.277,27.268,154.816
C04375=1074.226,228.810,-82.195,174.274,27.265,154.816
C04376=1074.220,228.561,-82.169,174.272,27.260,154.815
C04377=1074.214,228.313,-82.143,174.270,27.257,154.814
C04378=1074.208,228.064,-82.117,174.267,27.253,154.814
C04379=1074.203,227.815,-82.091,174.265,27.249,154.813
C04380=1074.197,227.567,-82.064,174.263,27.245,154.813
C04381=1074.191,227.318,-82.039,174.261,27.242,154.812
C04382=1074.185,227.070,-82.012,174.258,27.238,154.811
C04383=1074.180,226.821,-81.986,174.256,27.234,154.811
C04384=1074.173,226.573,-81.960,174.254,27.230,154.810
C04385=1074.168,226.324,-81.934,174.252,27.226,154.810
C04386=1074.162,226.075,-81.908,174.249,27.222,154.809
C04387=1074.156,225.828,-81.883,174.247,27.219,154.809
C04388=1074.151,225.579,-81.857,174.245,27.215,154.808
C04389=1074.145,225.330,-81.831,174.242,27.211,154.807
C04390=1074.139,225.082,-81.805,174.240,27.207,154.807
C04391=1074.133,224.833,-81.779,174.238,27.204,154.806
C04392=1074.127,224.584,-81.753,174.236,27.199,154.806
C04393=1074.121,224.336,-81.727,174.234,27.196,154.805
C04394=1074.116,224.087,-81.701,174.232,27.192,154.804
C04395=1074.110,223.838,-81.675,174.230,27.189,154.804
C04396=1074.104,223.590,-81.649,174.228,27.184,154.803
C04397=1074.099,223.341,-81.623,174.225,27.181,154.803
C04398=1074.093,223.093,-81.598,174.223,27.177,154.802
C04399=1074.083,222.673,-81.554,174.219,27.171,154.801
C04400=1074.074,222.253,-81.511,174.216,27.164,154.800
C04401=1074.064,221.833,-81.467,174.212,27.157,154.799
C04402=1074.054,221.414,-81.424,174.208,27.151,154.798
C04403=1074.049,221.165,-81.398,174.206,27.147,154.798
C04404=1074.043,220.916,-81.373,174.204,27.143,154.797
C04405=1074.036,220.667,-81.347,174.201,27.139,154.796
C04406=1074.031,220.418,-81.321,174.199,27.135,154.796
C04407=1074.025,220.170,-81.296,174.197,27.132,154.795
C04408=1074.019,219.921,-81.270,174.195,27.128,154.795
C04409=1074.014,219.673,-81.245,174.192,27.124,154.794
C04410=1074.007,219.424,-81.220,174.191,27.121,154.794
C04411=1074.002,219.176,-81.193,174.189,27.117,154.793
C04412=1073.995,218.927,-81.168,174.186,27.113,154.792
C04413=1073.989,218.678,-81.142,174.184,27.109,154.792
C04414=1073.984,218.430,-81.116,174.182,27.105,154.791
C04415=1073.978,218.182,-81.091,174.180,27.101,154.791
C04416=1073.973,217.933,-81.066,174.177,27.097,154.790
C04417=1073.967,217.683,-81.041,174.175,27.094,154.790
C04418=1073.961,217.435,-81.016,174.173,27.090,154.789
C04419=1073.956,217.186,-80.990,174.171,27.086,154.788
C04420=1073.949,216.938,-80.965,174.168,27.082,154.788
C04421=1073.943,216.689,-80.939,174.166,27.078,154.787
C04422=1073.938,216.440,-80.913,174.165,27.075,154.787
C04423=1073.932,216.192,-80.888,174.163,27.071,154.786
C04424=1073.926,215.943,-80.863,174.160,27.067,154.785
C04425=1073.920,215.694,-80.837,174.158,27.063,154.785
C04426=1073.914,215.446,-80.812,174.156,27.059,154.784
C04427=1073.909,215.197,-80.788,174.154,27.055,154.784
C04428=1073.903,214.948,-80.762,174.151,27.052,154.783
C04429=1073.897,214.699,-80.736,174.149,27.048,154.782
C04430=1073.892,214.452,-80.711,174.147,27.044,154.782
C04431=1073.886,214.203,-80.686,174.146,27.040,154.781
C04432=1073.880,213.954,-80.660,174.143,27.036,154.781
C04433=1073.874,213.705,-80.635,174.141,27.032,154.780
C04434=1073.869,213.457,-80.610,174.139,27.028,154.779
C04435=1073.863,213.208,-80.584,174.137,27.024,154.779
C04436=1073.857,212.959,-80.559,174.134,27.021,154.778
C04437=1073.852,212.710,-80.535,174.132,27.017,154.778
C04438=1073.845,212.462,-80.510,174.130,27.013,154.777
C04439=1073.839,212.213,-80.484,174.129,27.009,154.777
C04440=1073.834,211.964,-80.460,174.126,27.006,154.776
C04441=1073.828,211.715,-80.434,174.124,27.002,154.775
C04442=1073.822,211.467,-80.409,174.122,26.998,154.775
C04443=1073.817,211.218,-80.384,174.120,26.994,154.774
C04444=1073.811,210.970,-80.359,174.118,26.990,154.774
C04445=1073.804,210.721,-80.334,174.115,26.986,154.773
C04446=1073.799,210.472,-80.310,174.113,26.982,154.772
C04447=1073.793,210.224,-80.284,174.112,26.979,154.772
C04448=1073.788,209.975,-80.260,174.110,26.975,154.771
C04449=1073.781,209.726,-80.235,174.107,26.971,154.771
C04450=1073.776,209.477,-80.209,174.105,26.967,154.770
C04451=1073.766,209.063,-80.168,174.101,26.961,154.769
C04452=1073.757,208.647,-80.126,174.098,26.954,154.768
C04453=1073.747,208.231,-80.084,174.095,26.948,154.767
C04454=1073.737,207.816,-80.043,174.091,26.941,154.766
C04455=1073.713,206.776,-79.942,173.966,26.876,154.765
C04456=1073.707,206.527,-79.917,173.965,26.873,154.765
C04457=1073.702,206.278,-79.893,173.963,26.870,154.764
C04458=1073.697,206.030,-79.869,173.960,26.868,154.764
C04459=1073.691,205.781,-79.845,173.958,26.865,154.764
C04460=1073.685,205.531,-79.821,173.955,26.862,154.763
C04461=1073.680,205.283,-79.797,173.953,26.858,154.763
C04462=1073.674,205.034,-79.773,173.952,26.856,154.763
C04463=1073.668,204.785,-79.749,173.949,26.853,154.762
C04464=1073.663,204.537,-79.725,173.947,26.850,154.762
C04465=1073.657,204.288,-79.700,173.944,26.847,154.762
C04466=1073.651,204.040,-79.677,173.942,26.844,154.761
C04467=1073.645,203.791,-79.652,173.940,26.841,154.761
C04468=1073.640,203.541,-79.629,173.938,26.838,154.760
C04469=1073.634,203.293,-79.605,173.936,26.836,154.760
C04470=1073.629,203.045,-79.581,173.933,26.833,154.760
C04471=1073.623,202.795,-79.556,173.931,26.830,154.759
C04472=1073.618,202.547,-79.532,173.928,26.827,154.759
C04473=1073.612,202.298,-79.509,173.927,26.824,154.759
C04474=1073.607,202.049,-79.485,173.925,26.821,154.758
C04475=1073.600,201.800,-79.461,173.922,26.818,154.758
C04476=1073.595,201.552,-79.436,173.920,26.815,154.758
C04477=1073.589,201.303,-79.413,173.917,26.813,154.757
C04478=1073.582,201.054,-79.389,173.916,26.810,154.757
C04479=1073.577,200.805,-79.365,173.913,26.807,154.756
C04480=1073.571,200.556,-79.342,173.911,26.804,154.756
C04481=1073.566,200.308,-79.318,173.909,26.801,154.756
C04482=1073.559,200.059,-79.294,173.906,26.798,154.755
C04483=1073.554,199.809,-79.270,173.905,26.796,154.755
C04484=1073.548,199.561,-79.247,173.902,26.793,154.755
C04485=1073.543,199.312,-79.224,173.900,26.790,154.754
C04486=1073.537,199.064,-79.199,173.898,26.787,154.754
C04487=1073.531,198.815,-79.175,173.895,26.784,154.754
C04488=1073.526,198.565,-79.152,173.894,26.782,154.753
C04489=1073.520,198.317,-79.128,173.891,26.778,154.753
C04490=1073.515,198.068,-79.105,173.889,26.776,154.753
C04491=1073.508,197.819,-79.081,173.886,26.773,154.752
C04492=1073.502,197.571,-79.057,173.885,26.770,154.752
C04493=1073.497,197.322,-79.033,173.882,26.768,154.752
C04494=1073.491,197.073,-79.010,173.880,26.765,154.751
C04495=1073.486,196.824,-78.986,173.878,26.761,154.751
C04496=1073.480,196.576,-78.963,173.875,26.759,154.751
C04497=1073.474,196.326,-78.939,173.874,26.756,154.750
C04498=1073.468,196.078,-78.915,173.871,26.753,154.750
C04499=1073.463,195.829,-78.892,173.869,26.751,154.749
C04500=1073.457,195.580,-78.869,173.867,26.748,154.749
C04501=1073.452,195.331,-78.845,173.865,26.745,154.749
C04502=1073.446,195.082,-78.822,173.863,26.742,154.748
C04503=1073.441,194.834,-78.798,173.860,26.739,154.748
C04504=1073.435,194.585,-78.775,173.858,26.736,154.748
C04505=1073.428,194.336,-78.751,173.856,26.734,154.747
C04506=1073.423,194.087,-78.727,173.854,26.731,154.747
C04507=1073.417,193.838,-78.704,173.852,26.728,154.747
C04508=1073.411,193.589,-78.680,173.850,26.725,154.746
C04509=1073.406,193.340,-78.657,173.848,26.722,154.746
C04510=1073.401,193.091,-78.634,173.845,26.719,154.745
C04511=1073.395,192.843,-78.610,173.843,26.716,154.745
C04512=1073.390,192.594,-78.587,173.841,26.714,154.745
C04513=1073.384,192.345,-78.564,173.839,26.711,154.744
C04514=1073.378,192.097,-78.540,173.837,26.708,154.744
C04515=1073.373,191.848,-78.517,173.834,26.705,154.744
C04516=1073.366,191.566,-78.491,173.832,26.702,154.743
C04517=1073.359,191.285,-78.464,173.830,26.699,154.743
C04518=1073.354,191.004,-78.438,173.827,26.696,154.743
C04519=1073.347,190.722,-78.411,173.825,26.693,154.742
C04520=1073.342,190.473,-78.388,173.822,26.690,154.742
C04521=1073.335,190.225,-78.365,173.821,26.687,154.741
C04522=1073.331,189.976,-78.341,173.819,26.684,154.741
C04523=1073.325,189.727,-78.318,173.816,26.681,154.741
C04524=1073.319,189.478,-78.295,173.815,26.678,154.740
C04525=1073.314,189.229,-78.271,173.812,26.676,154.740
C04526=1073.308,188.980,-78.248,173.810,26.673,154.740
C04527=1073.302,188.732,-78.225,173.808,26.670,154.739
C04528=1073.297,188.483,-78.202,173.806,26.667,154.739
C04529=1073.292,188.233,-78.179,173.804,26.664,154.739
C04530=1073.286,187.985,-78.156,173.802,26.662,154.738
C04531=1073.280,187.736,-78.133,173.800,26.659,154.738
C04532=1073.274,187.487,-78.110,173.797,26.656,154.737
C04533=1073.269,187.238,-78.086,173.796,26.653,154.737
C04534=1073.264,186.990,-78.063,173.794,26.650,154.737
C04535=1073.258,186.741,-78.040,173.791,26.647,154.736
C04536=1073.252,186.492,-78.017,173.789,26.645,154.736
C04537=1073.247,186.243,-77.994,173.787,26.642,154.736
C04538=1073.242,185.994,-77.971,173.785,26.639,154.735
C04539=1073.236,185.745,-77.948,173.783,26.636,154.735
C04540=1073.230,185.496,-77.925,173.781,26.633,154.735
C04541=1073.225,185.247,-77.901,173.779,26.630,154.734
C04542=1073.220,184.998,-77.878,173.777,26.628,154.734
C04543=1073.214,184.749,-77.855,173.775,26.625,154.733
C04544=1073.208,184.500,-77.832,173.772,26.622,154.733
C04545=1073.202,184.251,-77.809,173.771,26.620,154.733
C04546=1073.197,184.003,-77.787,173.768,26.617,154.732
C04547=1073.190,183.754,-77.764,173.766,26.614,154.732
C04548=1073.184,183.505,-77.741,173.765,26.611,154.732
C04549=1073.179,183.256,-77.718,173.762,26.609,154.732
C04550=1073.173,183.007,-77.696,173.760,26.606,154.731
C04551=1073.168,182.758,-77.673,173.758,26.603,154.731
C04552=1073.161,182.509,-77.651,173.756,26.600,154.730
C04553=1073.155,182.260,-77.628,173.753,26.598,154.730
C04554=1073.150,182.011,-77.605,173.752,26.595,154.730
C04555=1073.144,181.763,-77.582,173.749,26.593,154.730
C04556=1073.139,181.514,-77.559,173.747,26.589,154.729
C04557=1073.133,181.265,-77.538,173.746,26.587,154.729
C04558=1073.127,181.016,-77.515,173.743,26.584,154.728
C04559=1073.121,180.767,-77.492,173.741,26.582,154.728
C04560=1073.115,180.518,-77.469,173.739,26.579,154.728
C04561=1073.110,180.270,-77.446,173.737,26.576,154.728
C04562=1073.104,180.020,-77.424,173.735,26.573,154.727
C04563=1073.098,179.771,-77.401,173.733,26.571,154.727
C04564=1073.092,179.523,-77.378,173.731,26.568,154.726
C04565=1073.086,179.274,-77.355,173.729,26.566,154.726
C04566=1073.080,179.024,-77.334,173.727,26.563,154.726
C04567=1073.075,178.776,-77.311,173.725,26.560,154.725
C04568=1073.069,178.527,-77.288,173.723,26.557,154.725
C04569=1073.064,178.278,-77.266,173.720,26.555,154.725
C04570=1073.057,178.029,-77.244,173.719,26.552,154.724
C04571=1073.052,177.780,-77.221,173.717,26.549,154.724
C04572=1073.046,177.531,-77.199,173.714,26.546,154.724
C04573=1073.041,177.282,-77.176,173.713,26.544,154.723
C04574=1073.035,177.034,-77.154,173.710,26.541,154.723
C04575=1073.029,176.784,-77.131,173.709,26.539,154.723
C04576=1073.023,176.536,-77.108,173.706,26.536,154.722
C04577=1073.018,176.287,-77.085,173.704,26.533,154.722
C04578=1073.012,176.037,-77.064,173.703,26.530,154.722
C04579=1073.006,175.789,-77.041,173.700,26.528,154.722
C04580=1073.000,175.507,-77.016,173.698,26.525,154.721
C04581=1072.993,175.226,-76.990,173.695,26.522,154.721
C04582=1072.987,174.943,-76.965,173.694,26.519,154.720
C04583=1072.981,174.662,-76.940,173.692,26.516,154.720
C04584=1072.975,174.413,-76.917,173.689,26.513,154.720
C04585=1072.969,174.164,-76.895,173.687,26.510,154.719
C04586=1072.964,173.916,-76.873,173.685,26.507,154.719
C04587=1072.958,173.666,-76.851,173.683,26.505,154.719
C04588=1072.952,173.418,-76.828,173.681,26.502,154.718
C04589=1072.946,173.168,-76.806,173.679,26.499,154.718
C04590=1072.941,172.920,-76.783,173.678,26.497,154.718
C04591=1072.935,172.671,-76.762,173.675,26.493,154.717
C04592=1072.929,172.422,-76.739,173.673,26.491,154.717
C04593=1072.924,172.172,-76.717,173.671,26.488,154.716
C04594=1072.918,171.924,-76.695,173.669,26.486,154.716
C04595=1072.912,171.675,-76.672,173.668,26.483,154.716
C04596=1072.907,171.426,-76.650,173.665,26.480,154.716
C04597=1072.901,171.177,-76.628,173.664,26.477,154.715
C04598=1072.896,170.928,-76.606,173.661,26.474,154.715
C04599=1072.890,170.679,-76.583,173.660,26.472,154.714
C04600=1072.884,170.430,-76.561,173.657,26.469,154.714
C04601=1072.879,170.182,-76.539,173.655,26.466,154.714
C04602=1072.873,169.932,-76.517,173.654,26.464,154.713
C04603=1072.867,169.683,-76.495,173.651,26.461,154.713
C04604=1072.862,169.435,-76.472,173.650,26.458,154.713
C04605=1072.857,169.185,-76.450,173.647,26.455,154.712
C04606=1072.850,168.936,-76.429,173.646,26.453,154.712
C04607=1072.845,168.688,-76.406,173.643,26.450,154.712
C04608=1072.839,168.439,-76.384,173.642,26.448,154.711
C04609=1072.834,168.189,-76.362,173.640,26.445,154.711
C04610=1072.829,167.940,-76.340,173.638,26.442,154.711
C04611=1072.822,167.692,-76.318,173.636,26.439,154.710
C04612=1072.818,167.443,-76.296,173.634,26.436,154.710
C04613=1072.812,167.193,-76.274,173.632,26.434,154.710
C04614=1072.806,166.944,-76.252,173.630,26.431,154.709
C04615=1072.801,166.696,-76.230,173.628,26.428,154.709
C04616=1072.795,166.447,-76.208,173.627,26.426,154.709
C04617=1072.790,166.198,-76.186,173.624,26.423,154.708
C04618=1072.784,165.949,-76.164,173.623,26.420,154.708
C04619=1072.778,165.699,-76.142,173.620,26.417,154.708
C04620=1072.773,165.451,-76.120,173.619,26.414,154.707
C04621=1072.767,165.202,-76.098,173.617,26.412,154.707
C04622=1072.762,164.953,-76.076,173.615,26.409,154.706
C04623=1072.756,164.704,-76.054,173.613,26.406,154.706
C04624=1072.751,164.455,-76.033,173.611,26.404,154.706
C04625=1072.746,164.205,-76.010,173.609,26.401,154.705
C04626=1072.740,163.958,-75.988,173.608,26.398,154.705
C04627=1072.735,163.708,-75.966,173.605,26.395,154.705
C04628=1072.729,163.460,-75.945,173.604,26.393,154.704
C04629=1072.724,163.210,-75.923,173.601,26.390,154.704
C04630=1072.718,162.962,-75.901,173.600,26.387,154.704
C04631=1072.713,162.712,-75.879,173.597,26.384,154.703
C04632=1072.707,162.464,-75.858,173.596,26.382,154.703
C04633=1072.702,162.214,-75.836,173.594,26.379,154.703
C04634=1072.696,161.965,-75.814,173.592,26.376,154.702
C04635=1072.691,161.716,-75.792,173.590,26.373,154.702
C04636=1072.686,161.467,-75.770,173.588,26.371,154.702
C04637=1072.680,161.218,-75.749,173.586,26.367,154.701
C04638=1072.673,160.969,-75.727,173.585,26.365,154.701
C04639=1072.668,160.720,-75.706,173.582,26.362,154.700
C04640=1072.662,160.471,-75.684,173.581,26.360,154.700
C04641=1072.657,160.222,-75.662,173.578,26.357,154.700
C04642=1072.651,159.973,-75.641,173.577,26.354,154.700
C04643=1072.645,159.725,-75.619,173.574,26.351,154.699
C04644=1072.639,159.442,-75.595,173.573,26.349,154.699
C04645=1072.632,159.160,-75.570,173.571,26.345,154.698
C04646=1072.626,158.878,-75.546,173.568,26.343,154.698
C04647=1072.619,158.596,-75.521,173.566,26.340,154.698
C04648=1072.614,158.347,-75.500,173.565,26.337,154.697
C04649=1072.608,158.098,-75.478,173.562,26.334,154.697
C04650=1072.602,157.849,-75.457,173.561,26.332,154.697
C04651=1072.596,157.600,-75.436,173.558,26.329,154.696
C04652=1072.591,157.351,-75.414,173.557,26.326,154.696
C04653=1072.585,157.102,-75.392,173.555,26.323,154.696
C04654=1072.580,156.853,-75.371,173.553,26.321,154.695
C04655=1072.574,156.604,-75.349,173.551,26.318,154.695
C04656=1072.568,156.355,-75.329,173.549,26.316,154.695
C04657=1072.563,156.105,-75.307,173.548,26.313,154.694
C04658=1072.557,155.857,-75.285,173.545,26.310,154.694
C04659=1072.551,155.608,-75.264,173.544,26.307,154.694
C04660=1072.546,155.359,-75.242,173.541,26.305,154.693
C04661=1072.540,155.109,-75.222,173.540,26.302,154.693
C04662=1072.534,154.861,-75.200,173.538,26.299,154.693
C04663=1072.529,154.612,-75.179,173.536,26.297,154.692
C04664=1072.522,154.363,-75.157,173.534,26.294,154.692
C04665=1072.517,154.114,-75.137,173.532,26.291,154.692
C04666=1072.512,153.864,-75.115,173.531,26.289,154.691
C04667=1072.506,153.616,-75.093,173.529,26.286,154.691
C04668=1072.500,153.366,-75.072,173.527,26.284,154.691
C04669=1072.495,153.118,-75.051,173.525,26.280,154.690
C04670=1072.489,152.868,-75.029,173.523,26.278,154.690
C04671=1072.483,152.619,-75.009,173.521,26.275,154.690
C04672=1072.478,152.371,-74.988,173.519,26.273,154.689
C04673=1072.472,152.121,-74.966,173.518,26.270,154.689
C04674=1072.466,151.872,-74.945,173.516,26.267,154.689
C04675=1072.460,151.623,-74.924,173.514,26.265,154.688
C04676=1072.455,151.375,-74.903,173.512,26.262,154.688
C04677=1072.449,151.125,-74.882,173.510,26.259,154.687
C04678=1072.443,150.876,-74.860,173.509,26.257,154.687
C04679=1072.438,150.627,-74.840,173.506,26.254,154.687
C04680=1072.432,150.378,-74.818,173.505,26.252,154.687
C04681=1072.427,150.129,-74.798,173.503,26.248,154.686
C04682=1072.420,149.880,-74.776,173.501,26.246,154.686
C04683=1072.415,149.631,-74.755,173.500,26.243,154.685
C04684=1072.410,149.382,-74.734,173.497,26.241,154.685
C04685=1072.403,149.133,-74.713,173.496,26.238,154.685
C04686=1072.398,148.884,-74.692,173.493,26.235,154.685
C04687=1072.393,148.635,-74.671,173.492,26.233,154.684
C04688=1072.387,148.385,-74.650,173.490,26.230,154.684
C04689=1072.381,148.137,-74.629,173.488,26.227,154.683
C04690=1072.376,147.888,-74.608,173.487,26.225,154.683
C04691=1072.369,147.639,-74.587,173.484,26.222,154.683
C04692=1072.364,147.390,-74.566,173.483,26.220,154.683
C04693=1072.358,147.140,-74.545,173.482,26.217,154.682
C04694=1072.352,146.891,-74.524,173.479,26.214,154.682
C04695=1072.347,146.642,-74.504,173.478,26.211,154.681
C04696=1072.341,146.393,-74.482,173.475,26.209,154.681
C04697=1072.335,146.144,-74.462,173.474,26.206,154.681
C04698=1072.329,145.896,-74.441,173.472,26.204,154.680
C04699=1072.324,145.646,-74.420,173.470,26.201,154.680
C04700=1072.318,145.397,-74.399,173.469,26.198,154.680
C04701=1072.313,145.148,-74.378,173.466,26.195,154.679
C04702=1072.306,144.899,-74.358,173.465,26.193,154.679
C04703=1072.301,144.650,-74.337,173.463,26.190,154.679
C04704=1072.295,144.401,-74.316,173.461,26.188,154.678
C04705=1072.289,144.151,-74.295,173.460,26.185,154.678
C04706=1072.284,143.902,-74.274,173.458,26.183,154.678
C04707=1072.278,143.654,-74.254,173.456,26.179,154.677
C04708=1072.272,143.371,-74.230,173.453,26.176,154.677
C04709=1072.265,143.089,-74.207,173.452,26.173,154.677
C04710=1072.258,142.807,-74.183,173.450,26.170,154.676
C04711=1072.253,142.524,-74.160,173.447,26.167,154.676
C04712=1072.247,142.275,-74.138,173.446,26.165,154.676
C04713=1072.241,142.027,-74.118,173.444,26.162,154.675
C04714=1072.235,141.777,-74.098,173.442,26.160,154.675
C04715=1072.230,141.528,-74.077,173.441,26.157,154.674
C04716=1072.224,141.279,-74.056,173.439,26.154,154.674
C04717=1072.218,141.030,-74.036,173.437,26.151,154.674
C04718=1072.212,140.781,-74.015,173.435,26.149,154.674
C04719=1072.207,140.531,-73.994,173.434,26.146,154.673
C04720=1072.201,140.283,-73.974,173.432,26.144,154.673
C04721=1072.196,140.034,-73.953,173.430,26.141,154.672
C04722=1072.190,139.784,-73.932,173.429,26.139,154.672
C04723=1072.184,139.535,-73.912,173.426,26.135,154.672
C04724=1072.179,139.286,-73.892,173.425,26.133,154.672
C04725=1072.173,139.037,-73.871,173.423,26.130,154.671
C04726=1072.167,138.788,-73.851,173.421,26.128,154.671
C04727=1072.161,138.539,-73.830,173.420,26.125,154.670
C04728=1072.155,138.290,-73.810,173.417,26.122,154.670
C04729=1072.150,138.041,-73.789,173.416,26.120,154.670
C04730=1072.144,137.791,-73.768,173.414,26.117,154.669
C04731=1072.138,137.543,-73.748,173.412,26.114,154.669
C04732=1072.133,137.293,-73.728,173.411,26.112,154.669
C04733=1072.127,137.045,-73.708,173.409,26.109,154.668
C04734=1072.122,136.796,-73.687,173.407,26.106,154.668
C04735=1072.115,136.546,-73.667,173.405,26.104,154.668
C04736=1072.110,136.297,-73.646,173.404,26.101,154.667
C04737=1072.104,136.048,-73.626,173.402,26.098,154.667
C04738=1072.098,135.799,-73.606,173.400,26.096,154.667
C04739=1072.093,135.550,-73.585,173.399,26.093,154.666
C04740=1072.087,135.300,-73.565,173.397,26.091,154.666
C04741=1072.081,135.051,-73.544,173.395,26.088,154.666
C04742=1072.075,134.802,-73.524,173.393,26.085,154.665
C04743=1072.070,134.553,-73.504,173.392,26.083,154.665
C04744=1072.064,134.304,-73.484,173.390,26.079,154.665
C04745=1072.059,134.055,-73.463,173.388,26.077,154.664
C04746=1072.052,133.806,-73.443,173.387,26.074,154.664
C04747=1072.047,133.557,-73.422,173.384,26.072,154.664
C04748=1072.041,133.308,-73.402,173.383,26.069,154.663
C04749=1072.036,133.059,-73.382,173.382,26.067,154.663
C04750=1072.030,132.810,-73.362,173.379,26.064,154.663
C04751=1072.025,132.560,-73.342,173.378,26.061,154.662
C04752=1072.019,132.311,-73.322,173.376,26.058,154.662
C04753=1072.013,132.062,-73.301,173.374,26.056,154.662
C04754=1072.007,131.813,-73.281,173.373,26.053,154.661
C04755=1072.001,131.564,-73.261,173.371,26.051,154.661
C04756=1071.996,131.315,-73.241,173.370,26.048,154.661
C04757=1071.990,131.066,-73.221,173.367,26.045,154.660
C04758=1071.984,130.817,-73.201,173.366,26.042,154.660
C04759=1071.977,130.567,-73.181,173.364,26.040,154.660
C04760=1071.972,130.318,-73.161,173.362,26.038,154.659
C04761=1071.966,130.069,-73.141,173.361,26.035,154.659
C04762=1071.960,129.820,-73.121,173.359,26.032,154.659
C04763=1071.954,129.571,-73.101,173.357,26.029,154.658
C04764=1071.949,129.322,-73.081,173.355,26.027,154.658
C04765=1071.943,129.073,-73.061,173.354,26.024,154.658
C04766=1071.937,128.823,-73.041,173.352,26.022,154.657
C04767=1071.931,128.574,-73.021,173.350,26.019,154.657
C04768=1071.926,128.325,-73.001,173.349,26.017,154.657
C04769=1071.920,128.076,-72.981,173.347,26.014,154.656
C04770=1071.914,127.827,-72.961,173.345,26.011,154.656
C04771=1071.908,127.578,-72.942,173.343,26.009,154.656
C04772=1071.902,127.296,-72.919,173.341,26.006,154.655
C04773=1071.895,127.012,-72.896,173.340,26.003,154.655
C04774=1071.888,126.730,-72.874,173.337,26.000,154.655
C04775=1071.882,126.448,-72.851,173.336,25.997,154.654
C04776=1071.876,126.199,-72.831,173.334,25.994,154.654
C04777=1071.871,125.950,-72.811,173.332,25.991,154.653
C04778=1071.865,125.701,-72.791,173.331,25.989,154.653
C04779=1071.859,125.452,-72.771,173.329,25.986,154.653
C04780=1071.853,125.203,-72.752,173.327,25.983,154.652
C04781=1071.847,124.954,-72.732,173.326,25.981,154.652
C04782=1071.842,124.704,-72.712,173.324,25.978,154.652
C04783=1071.835,124.454,-72.692,173.323,25.976,154.651
C04784=1071.829,124.206,-72.672,173.320,25.973,154.651
C04785=1071.824,123.956,-72.653,173.319,25.970,154.651
C04786=1071.818,123.707,-72.633,173.318,25.968,154.650
C04787=1071.813,123.458,-72.613,173.315,25.965,154.650
C04788=1071.807,123.209,-72.593,173.314,25.962,154.650
C04789=1071.801,122.959,-72.574,173.312,25.960,154.649
C04790=1071.795,122.711,-72.554,173.311,25.957,154.649
C04791=1071.789,122.462,-72.534,173.309,25.954,154.649
C04792=1071.783,122.212,-72.515,173.307,25.952,154.648
C04793=1071.778,121.963,-72.494,173.306,25.949,154.648
C04794=1071.773,121.714,-72.475,173.304,25.946,154.648
C04795=1071.767,121.465,-72.455,173.302,25.943,154.647
C04796=1071.761,121.216,-72.436,173.301,25.941,154.647
C04797=1071.755,120.967,-72.416,173.299,25.938,154.647
C04798=1071.750,120.718,-72.397,173.298,25.936,154.646
C04799=1071.744,120.469,-72.378,173.295,25.933,154.646
C04800=1071.739,120.219,-72.357,173.294,25.930,154.646
C04801=1071.733,119.970,-72.338,173.293,25.928,154.645
C04802=1071.727,119.721,-72.318,173.291,25.925,154.645
C04803=1071.721,119.472,-72.299,173.289,25.922,154.645
C04804=1071.715,119.223,-72.279,173.287,25.919,154.644
C04805=1071.710,118.974,-72.259,173.286,25.916,154.644
C04806=1071.704,118.724,-72.240,173.285,25.914,154.643
C04807=1071.698,118.475,-72.220,173.282,25.911,154.643
C04808=1071.693,118.226,-72.200,173.281,25.909,154.643
C04809=1071.687,117.977,-72.180,173.279,25.906,154.642
C04810=1071.681,117.727,-72.161,173.278,25.903,154.642
C04811=1071.676,117.479,-72.142,173.277,25.901,154.642
C04812=1071.670,117.230,-72.122,173.274,25.898,154.641
C04813=1071.665,116.980,-72.103,173.273,25.895,154.641
C04814=1071.659,116.731,-72.084,173.271,25.893,154.641
C04815=1071.653,116.482,-72.064,173.270,25.890,154.640
C04816=1071.647,116.233,-72.045,173.268,25.887,154.640
C04817=1071.642,115.983,-72.025,173.266,25.884,154.640
C04818=1071.637,115.733,-72.006,173.265,25.881,154.639
C04819=1071.631,115.485,-71.986,173.264,25.879,154.639
C04820=1071.626,115.236,-71.967,173.261,25.876,154.638
C04821=1071.620,114.987,-71.947,173.260,25.873,154.638
C04822=1071.614,114.738,-71.928,173.258,25.871,154.638
C04823=1071.608,114.488,-71.908,173.257,25.868,154.637
C04824=1071.603,114.239,-71.889,173.256,25.866,154.637
C04825=1071.597,113.989,-71.870,173.253,25.863,154.637
C04826=1071.592,113.741,-71.851,173.252,25.860,154.636
C04827=1071.586,113.492,-71.831,173.250,25.857,154.636
C04828=1071.580,113.242,-71.812,173.249,25.855,154.636
C04829=1071.574,112.993,-71.793,173.247,25.852,154.635
C04830=1071.568,112.744,-71.774,173.245,25.849,154.635
C04831=1071.562,112.494,-71.755,173.244,25.847,154.635
C04832=1071.556,112.246,-71.735,173.242,25.844,154.634
C04833=1071.551,111.997,-71.716,173.241,25.842,154.634
C04834=1071.546,111.747,-71.696,173.239,25.838,154.634
C04835=1071.540,111.498,-71.677,173.237,25.836,154.633
C04836=1071.533,111.215,-71.656,173.236,25.833,154.633
C04837=1071.526,110.933,-71.634,173.234,25.830,154.632
C04838=1071.519,110.651,-71.612,173.232,25.827,154.632
C04839=1071.513,110.368,-71.591,173.230,25.824,154.632
C04840=1071.507,110.119,-71.572,173.229,25.821,154.631
C04841=1071.501,109.869,-71.553,173.227,25.818,154.631
C04842=1071.496,109.620,-71.533,173.226,25.816,154.631
C04843=1071.490,109.371,-71.515,173.224,25.813,154.630
C04844=1071.484,109.122,-71.496,173.222,25.811,154.630
C04845=1071.479,108.873,-71.477,173.221,25.808,154.630
C04846=1071.473,108.623,-71.457,173.219,25.806,154.629
C04847=1071.466,108.374,-71.439,173.218,25.803,154.629
C04848=1071.460,108.125,-71.419,173.215,25.800,154.629
C04849=1071.455,107.876,-71.400,173.214,25.797,154.628
C04850=1071.449,107.627,-71.381,173.213,25.795,154.628
C04851=1071.444,107.377,-71.363,173.211,25.792,154.628
C04852=1071.438,107.128,-71.343,173.210,25.789,154.627
C04853=1071.432,106.878,-71.324,173.208,25.787,154.627
C04854=1071.426,106.630,-71.306,173.206,25.784,154.627
C04855=1071.421,106.381,-71.287,173.205,25.782,154.626
C04856=1071.415,106.131,-71.267,173.203,25.779,154.626
C04857=1071.409,105.882,-71.249,173.202,25.776,154.626
C04858=1071.403,105.633,-71.230,173.200,25.773,154.625
C04859=1071.398,105.384,-71.211,173.198,25.770,154.625
C04860=1071.391,105.135,-71.192,173.197,25.768,154.624
C04861=1071.386,104.885,-71.173,173.195,25.765,154.624
C04862=1071.381,104.637,-71.154,173.194,25.763,154.624
C04863=1071.374,104.387,-71.135,173.193,25.760,154.623
C04864=1071.368,104.138,-71.116,173.190,25.757,154.623
C04865=1071.363,103.888,-71.097,173.189,25.755,154.623
C04866=1071.357,103.640,-71.079,173.188,25.752,154.622
C04867=1071.352,103.390,-71.060,173.186,25.749,154.622
C04868=1071.346,103.141,-71.041,173.185,25.747,154.622
C04869=1071.339,102.892,-71.022,173.182,25.743,154.621
C04870=1071.334,102.643,-71.003,173.181,25.741,154.621
C04871=1071.329,102.393,-70.985,173.180,25.738,154.621
C04872=1071.323,102.144,-70.966,173.178,25.736,154.620
C04873=1071.317,101.895,-70.947,173.177,25.733,154.620
C04874=1071.312,101.645,-70.928,173.175,25.730,154.619
C04875=1071.305,101.396,-70.909,173.173,25.728,154.619
C04876=1071.301,101.147,-70.891,173.172,25.725,154.619
C04877=1071.294,100.898,-70.872,173.170,25.722,154.618
C04878=1071.288,100.648,-70.853,173.169,25.720,154.618
C04879=1071.282,100.399,-70.835,173.168,25.717,154.618
C04880=1071.277,100.150,-70.816,173.166,25.714,154.617
C04881=1071.271,99.901,-70.798,173.164,25.711,154.617
C04882=1071.265,99.651,-70.778,173.162,25.709,154.617
C04883=1071.259,99.403,-70.760,173.161,25.706,154.616
C04884=1071.253,99.153,-70.742,173.160,25.704,154.616
C04885=1071.247,98.904,-70.723,173.158,25.701,154.616
C04886=1071.241,98.655,-70.704,173.157,25.699,154.615
C04887=1071.236,98.405,-70.686,173.154,25.696,154.615
C04888=1071.230,98.156,-70.668,173.153,25.693,154.615
C04889=1071.224,97.907,-70.648,173.152,25.690,154.614
C04890=1071.219,97.658,-70.631,173.150,25.688,154.614
C04891=1071.212,97.409,-70.612,173.149,25.685,154.614
C04892=1071.207,97.159,-70.594,173.148,25.682,154.613
C04893=1071.201,96.910,-70.575,173.145,25.680,154.613
C04894=1071.195,96.661,-70.556,173.144,25.677,154.613
C04895=1071.189,96.411,-70.538,173.142,25.674,154.612
C04896=1071.184,96.162,-70.519,173.141,25.672,154.612
C04897=1071.178,95.913,-70.501,173.140,25.669,154.611
C04898=1071.172,95.663,-70.483,173.138,25.667,154.611
C04899=1071.166,95.415,-70.464,173.136,25.663,154.611
C04900=1071.159,95.132,-70.444,173.135,25.660,154.610
C04901=1071.153,94.850,-70.423,173.133,25.658,154.610
C04902=1071.147,94.567,-70.401,173.131,25.654,154.610
C04903=1071.140,94.285,-70.380,173.130,25.652,154.609
C04904=1071.134,94.036,-70.362,173.128,25.649,154.609
C04905=1071.128,93.786,-70.344,173.126,25.646,154.608
C04906=1071.123,93.537,-70.326,173.125,25.643,154.608
C04907=1071.117,93.288,-70.307,173.123,25.640,154.608
C04908=1071.111,93.038,-70.288,173.122,25.638,154.607
C04909=1071.106,92.789,-70.270,173.120,25.635,154.607
C04910=1071.099,92.540,-70.252,173.119,25.632,154.607
C04911=1071.094,92.291,-70.233,173.118,25.630,154.606
C04912=1071.088,92.041,-70.215,173.115,25.627,154.606
C04913=1071.083,91.792,-70.198,173.114,25.624,154.606
C04914=1071.077,91.543,-70.179,173.113,25.622,154.605
C04915=1071.071,91.294,-70.161,173.111,25.619,154.605
C04916=1071.065,91.045,-70.142,173.110,25.616,154.604
C04917=1071.060,90.795,-70.124,173.108,25.614,154.604
C04918=1071.054,90.546,-70.106,173.107,25.611,154.604
C04919=1071.048,90.296,-70.088,173.105,25.608,154.604
C04920=1071.042,90.047,-70.070,173.103,25.605,154.603
C04921=1071.036,89.798,-70.051,173.102,25.603,154.603
C04922=1071.030,89.548,-70.033,173.101,25.600,154.602
C04923=1071.025,89.299,-70.015,173.099,25.598,154.602
C04924=1071.018,89.050,-69.997,173.098,25.595,154.602
C04925=1071.013,88.801,-69.979,173.096,25.592,154.601
C04926=1071.007,88.551,-69.961,173.094,25.589,154.601
C04927=1071.001,88.303,-69.943,173.093,25.587,154.601
C04928=1070.995,88.053,-69.925,173.091,25.584,154.600
C04929=1070.989,87.803,-69.907,173.090,25.581,154.600
C04930=1070.984,87.555,-69.888,173.089,25.579,154.600
C04931=1070.978,87.305,-69.870,173.087,25.576,154.599
C04932=1070.972,87.056,-69.853,173.086,25.574,154.599
C04933=1070.966,86.807,-69.834,173.084,25.571,154.599
C04934=1070.960,86.558,-69.816,173.082,25.568,154.598
C04935=1070.954,86.308,-69.798,173.081,25.566,154.598
C04936=1070.948,86.059,-69.781,173.079,25.563,154.598
C04937=1070.942,85.810,-69.762,173.078,25.560,154.597
C04938=1070.936,85.561,-69.745,173.077,25.558,154.597
C04939=1070.931,85.311,-69.726,173.075,25.555,154.596
C04940=1070.926,85.062,-69.709,173.074,25.552,154.596
C04941=1070.919,84.812,-69.691,173.072,25.549,154.596
C04942=1070.914,84.563,-69.672,173.070,25.547,154.596
C04943=1070.908,84.314,-69.654,173.069,25.544,154.595
C04944=1070.902,84.065,-69.637,173.067,25.541,154.595
C04945=1070.896,83.815,-69.619,173.066,25.539,154.594
C04946=1070.890,83.566,-69.601,173.065,25.536,154.594
C04947=1070.884,83.317,-69.583,173.063,25.533,154.594
C04948=1070.878,83.068,-69.565,173.062,25.531,154.593
C04949=1070.872,82.818,-69.547,173.061,25.528,154.593
C04950=1070.867,82.569,-69.530,173.058,25.525,154.593
C04951=1070.861,82.319,-69.512,173.057,25.522,154.592
C04952=1070.856,82.070,-69.494,173.056,25.520,154.592
C04953=1070.850,81.821,-69.476,173.054,25.517,154.592
C04954=1070.844,81.571,-69.458,173.053,25.514,154.591
C04955=1070.838,81.323,-69.440,173.051,25.511,154.591
C04956=1070.832,81.073,-69.422,173.050,25.509,154.591
C04957=1070.827,80.824,-69.404,173.049,25.506,154.590
C04958=1070.821,80.574,-69.386,173.047,25.503,154.590
C04959=1070.815,80.325,-69.369,173.045,25.501,154.589
C04960=1070.810,80.076,-69.351,173.044,25.498,154.589
C04961=1070.804,79.826,-69.333,173.042,25.495,154.589
C04962=1070.798,79.577,-69.316,173.041,25.493,154.588
C04963=1070.792,79.328,-69.298,173.040,25.490,154.588
C04964=1070.785,79.045,-69.278,173.038,25.487,154.588
C04965=1070.779,78.763,-69.258,173.036,25.484,154.587
C04966=1070.773,78.481,-69.237,173.035,25.481,154.587
C04967=1070.766,78.198,-69.217,173.032,25.478,154.586
C04968=1070.760,77.949,-69.200,173.031,25.475,154.586
C04969=1070.754,77.699,-69.182,173.030,25.472,154.586
C04970=1070.748,77.450,-69.164,173.028,25.470,154.585
C04971=1070.742,77.202,-69.147,173.027,25.467,154.585
C04972=1070.736,76.951,-69.130,173.026,25.464,154.585
C04973=1070.731,76.702,-69.113,173.024,25.462,154.584
C04974=1070.725,76.453,-69.095,173.023,25.459,154.584
C04975=1070.719,76.204,-69.077,173.021,25.456,154.584
C04976=1070.714,75.954,-69.059,173.020,25.453,154.583
C04977=1070.707,75.705,-69.042,173.018,25.451,154.583
C04978=1070.701,75.456,-69.025,173.016,25.448,154.583
C04979=1070.695,75.206,-69.007,173.015,25.446,154.582
C04980=1070.690,74.957,-68.989,173.014,25.443,154.582
C04981=1070.684,74.708,-68.972,173.012,25.440,154.581
C04982=1070.678,74.458,-68.955,173.011,25.438,154.581
C04983=1070.672,74.209,-68.937,173.010,25.435,154.581
C04984=1070.667,73.960,-68.920,173.008,25.432,154.580
C04985=1070.660,73.710,-68.902,173.007,25.430,154.580
C04986=1070.655,73.461,-68.884,173.005,25.427,154.580
C04987=1070.649,73.213,-68.867,173.003,25.424,154.579
C04988=1070.643,72.962,-68.850,173.002,25.421,154.579
C04989=1070.637,72.713,-68.833,173.000,25.418,154.579
C04990=1070.632,72.464,-68.815,172.999,25.416,154.578
C04991=1070.625,72.215,-68.798,172.998,25.413,154.578
C04992=1070.619,71.966,-68.780,172.996,25.411,154.578
C04993=1070.614,71.716,-68.763,172.995,25.408,154.577
C04994=1070.608,71.466,-68.745,172.994,25.405,154.577
C04995=1070.602,71.218,-68.728,172.992,25.403,154.577
C04996=1070.596,70.968,-68.711,172.991,25.400,154.576
C04997=1070.591,70.718,-68.694,172.990,25.397,154.576
C04998=1070.585,70.469,-68.676,172.987,25.394,154.575
C04999=1070.579,70.220,-68.659,172.986,25.391,154.575
C05000=1070.573,69.971,-68.641,172.984,25.389,154.575
C05001=1070.567,69.721,-68.624,172.983,25.386,154.574
C05002=1070.561,69.472,-68.607,172.982,25.383,154.574
C05003=1070.556,69.223,-68.590,172.980,25.381,154.574
C05004=1070.550,68.973,-68.572,172.979,25.378,154.573
C05005=1070.544,68.724,-68.555,172.978,25.376,154.573
C05006=1070.538,68.475,-68.538,172.976,25.373,154.573
C05007=1070.532,68.225,-68.521,172.975,25.370,154.572
C05008=1070.526,67.976,-68.504,172.974,25.368,154.572
C05009=1070.520,67.727,-68.486,172.971,25.364,154.572
C05010=1070.515,67.477,-68.469,172.970,25.362,154.571
C05011=1070.508,67.228,-68.452,172.969,25.359,154.571
C05012=1070.503,66.979,-68.434,172.967,25.356,154.570
C05013=1070.497,66.729,-68.418,172.966,25.354,154.570
C05014=1070.491,66.480,-68.400,172.964,25.351,154.570
C05015=1070.485,66.230,-68.384,172.963,25.349,154.569
C05016=1070.479,65.981,-68.366,172.962,25.346,154.569
C05017=1070.474,65.732,-68.349,172.960,25.343,154.569
C05018=1070.467,65.482,-68.332,172.959,25.341,154.568
C05019=1070.462,65.233,-68.315,172.958,25.338,154.568
C05020=1070.456,64.984,-68.298,172.956,25.336,154.568
C05021=1070.450,64.735,-68.281,172.954,25.332,154.567
C05022=1070.444,64.485,-68.264,172.953,25.329,154.567
C05023=1070.438,64.236,-68.247,172.951,25.327,154.567
C05024=1070.432,63.986,-68.230,172.950,25.324,154.566
C05025=1070.427,63.737,-68.213,172.949,25.322,154.566
C05026=1070.420,63.487,-68.196,172.947,25.319,154.566
C05027=1070.414,63.239,-68.179,172.946,25.317,154.565
C05028=1070.408,62.956,-68.160,172.944,25.314,154.565
C05029=1070.400,62.674,-68.141,172.942,25.311,154.565
C05030=1070.394,62.390,-68.122,172.941,25.308,154.564
C05031=1070.387,62.108,-68.102,172.940,25.305,154.564
C05032=1070.381,61.859,-68.086,172.938,25.302,154.563
C05033=1070.375,61.610,-68.069,172.936,25.299,154.563
C05034=1070.370,61.360,-68.052,172.935,25.296,154.563
C05035=1070.363,61.111,-68.035,172.933,25.294,154.562
C05036=1070.357,60.861,-68.018,172.932,25.291,154.562
C05037=1070.352,60.612,-68.002,172.930,25.289,154.562
C05038=1070.345,60.363,-67.985,172.929,25.286,154.561
C05039=1070.339,60.113,-67.968,172.928,25.284,154.561
C05040=1070.333,59.864,-67.950,172.926,25.281,154.561
C05041=1070.327,59.615,-67.934,172.925,25.278,154.560
C05042=1070.321,59.365,-67.918,172.924,25.275,154.560
C05043=1070.315,59.117,-67.901,172.922,25.273,154.560
C05044=1070.309,58.866,-67.884,172.921,25.270,154.559
C05045=1070.303,58.617,-67.867,172.920,25.268,154.559
C05046=1070.297,58.368,-67.850,172.917,25.265,154.559
C05047=1070.292,58.118,-67.834,172.916,25.262,154.558
C05048=1070.286,57.869,-67.817,172.915,25.259,154.558
C05049=1070.279,57.620,-67.800,172.913,25.257,154.558
C05050=1070.274,57.370,-67.783,172.912,25.254,154.557
C05051=1070.268,57.121,-67.767,172.911,25.251,154.557
C05052=1070.262,56.871,-67.751,172.909,25.249,154.557
C05053=1070.256,56.623,-67.734,172.908,25.246,154.556
C05054=1070.251,56.373,-67.717,172.906,25.244,154.556
C05055=1070.245,56.124,-67.701,172.905,25.241,154.555
C05056=1070.238,55.874,-67.683,172.904,25.238,154.555
C05057=1070.233,55.624,-67.666,172.902,25.236,154.555
C05058=1070.227,55.375,-67.650,172.901,25.233,154.554
C05059=1070.221,55.126,-67.634,172.900,25.230,154.554
C05060=1070.215,54.876,-67.618,172.898,25.228,154.554
C05061=1070.209,54.627,-67.600,172.896,25.225,154.553
C05062=1070.203,54.378,-67.584,172.895,25.222,154.553
C05063=1070.197,54.129,-67.568,172.893,25.219,154.553
C05064=1070.191,53.879,-67.551,172.892,25.217,154.552
C05065=1070.186,53.629,-67.534,172.891,25.214,154.552
C05066=1070.179,53.380,-67.517,172.889,25.212,154.552
C05067=1070.173,53.131,-67.501,172.888,25.209,154.551
C05068=1070.167,52.882,-67.485,172.887,25.206,154.551
C05069=1070.162,52.632,-67.468,172.885,25.203,154.551
C05070=1070.156,52.383,-67.451,172.884,25.201,154.550
C05071=1070.150,52.133,-67.435,172.882,25.198,154.550
C05072=1070.144,51.884,-67.418,172.881,25.195,154.549
C05073=1070.139,51.635,-67.401,172.880,25.192,154.549
C05074=1070.133,51.385,-67.385,172.878,25.190,154.549
C05075=1070.127,51.136,-67.369,172.877,25.187,154.548
C05076=1070.121,50.887,-67.353,172.876,25.185,154.548
C05077=1070.115,50.637,-67.336,172.874,25.182,154.548
C05078=1070.110,50.388,-67.320,172.872,25.179,154.547
C05079=1070.104,50.138,-67.303,172.871,25.176,154.547
C05080=1070.097,49.888,-67.287,172.869,25.174,154.547
C05081=1070.091,49.639,-67.270,172.868,25.171,154.546
C05082=1070.085,49.390,-67.254,172.867,25.168,154.546
C05083=1070.080,49.140,-67.237,172.865,25.165,154.546
C05084=1070.074,48.891,-67.221,172.864,25.163,154.545
C05085=1070.068,48.641,-67.205,172.863,25.160,154.545
C05086=1070.062,48.392,-67.189,172.861,25.158,154.545
C05087=1070.056,48.143,-67.172,172.860,25.155,154.544
C05088=1070.051,47.893,-67.155,172.859,25.152,154.544
C05089=1070.045,47.644,-67.139,172.857,25.150,154.544
C05090=1070.040,47.395,-67.123,172.856,25.147,154.543
C05091=1070.034,47.146,-67.107,172.855,25.144,154.543
C05092=1070.028,46.863,-67.088,172.852,25.141,154.542
C05093=1070.021,46.580,-67.070,172.851,25.138,154.542
C05094=1070.014,46.298,-67.051,172.850,25.135,154.542
C05095=1070.008,46.015,-67.032,172.848,25.132,154.541
C05096=1070.002,45.765,-67.016,172.846,25.129,154.541
C05097=1069.996,45.516,-67.000,172.845,25.126,154.541
C05098=1069.990,45.266,-66.984,172.844,25.123,154.540
C05099=1069.985,45.017,-66.967,172.842,25.121,154.540
C05100=1069.979,44.767,-66.951,172.841,25.118,154.539
C05101=1069.973,44.518,-66.935,172.840,25.115,154.539
C05102=1069.967,44.268,-66.919,172.838,25.112,154.539
C05103=1069.961,44.019,-66.902,172.837,25.110,154.538
C05104=1069.955,43.770,-66.886,172.836,25.107,154.538
C05105=1069.949,43.520,-66.870,172.834,25.104,154.538
C05106=1069.943,43.270,-66.854,172.833,25.102,154.537
C05107=1069.937,43.021,-66.838,172.832,25.099,154.537
C05108=1069.932,42.772,-66.822,172.830,25.097,154.537
C05109=1069.926,42.522,-66.806,172.829,25.094,154.536
C05110=1069.920,42.273,-66.789,172.828,25.091,154.536
C05111=1069.914,42.024,-66.773,172.826,25.089,154.536
C05112=1069.909,41.774,-66.758,172.825,25.086,154.535
C05113=1069.903,41.525,-66.742,172.824,25.083,154.535
C05114=1069.897,41.276,-66.725,172.821,25.081,154.535
C05115=1069.891,41.026,-66.709,172.820,25.078,154.534
C05116=1069.885,40.777,-66.693,172.819,25.075,154.534
C05117=1069.879,40.527,-66.677,172.817,25.073,154.534
C05118=1069.873,40.278,-66.661,172.816,25.070,154.533
C05119=1069.867,40.029,-66.645,172.814,25.067,154.533
C05120=1069.861,39.779,-66.629,172.813,25.064,154.532
C05121=1069.855,39.529,-66.614,172.812,25.062,154.532
C05122=1069.849,39.280,-66.597,172.810,25.059,154.532
C05123=1069.844,39.031,-66.581,172.809,25.057,154.531
C05124=1069.838,38.781,-66.566,172.808,25.054,154.531
C05125=1069.832,38.532,-66.550,172.807,25.051,154.531
C05126=1069.826,38.283,-66.533,172.805,25.049,154.530
C05127=1069.820,38.033,-66.517,172.804,25.046,154.530
C05128=1069.814,37.783,-66.502,172.802,25.043,154.530
C05129=1069.808,37.534,-66.486,172.801,25.040,154.529
C05130=1069.802,37.285,-66.470,172.800,25.038,154.529
C05131=1069.796,37.035,-66.454,172.798,25.035,154.529
C05132=1069.791,36.786,-66.438,172.797,25.033,154.528
C05133=1069.784,36.537,-66.423,172.796,25.030,154.528
C05134=1069.779,36.287,-66.407,172.794,25.028,154.528
C05135=1069.773,36.038,-66.391,172.793,25.025,154.527
C05136=1069.767,35.788,-66.375,172.791,25.022,154.527
C05137=1069.760,35.539,-66.360,172.789,25.019,154.527
C05138=1069.755,35.289,-66.344,172.788,25.017,154.526
C05139=1069.749,35.040,-66.328,172.787,25.014,154.526
C05140=1069.743,34.790,-66.312,172.785,25.011,154.526
C05141=1069.737,34.541,-66.297,172.784,25.009,154.525
C05142=1069.731,34.292,-66.281,172.783,25.006,154.525
C05143=1069.725,34.042,-66.265,172.781,25.003,154.525
C05144=1069.719,33.793,-66.249,172.780,25.001,154.524
C05145=1069.713,33.543,-66.234,172.779,24.998,154.524
C05146=1069.707,33.294,-66.218,172.777,24.996,154.524
C05147=1069.701,33.044,-66.203,172.776,24.993,154.523
C05148=1069.695,32.795,-66.187,172.774,24.990,154.523
C05149=1069.690,32.545,-66.171,172.773,24.988,154.523
C05150=1069.684,32.296,-66.155,172.772,24.985,154.522
C05151=1069.677,32.046,-66.140,172.770,24.983,154.522
C05152=1069.671,31.797,-66.124,172.769,24.980,154.522
C05153=1069.666,31.548,-66.109,172.768,24.978,154.521
C05154=1069.660,31.299,-66.093,172.766,24.975,154.521
C05155=1069.654,31.049,-66.077,172.765,24.972,154.520
C05156=1069.647,30.766,-66.059,172.763,24.969,154.520
C05157=1069.640,30.483,-66.041,172.762,24.966,154.520
C05158=1069.634,30.201,-66.024,172.760,24.963,154.519
C05159=1069.627,29.918,-66.007,172.758,24.960,154.519
C05160=1069.621,29.669,-65.991,172.757,24.957,154.519
C05161=1069.615,29.419,-65.975,172.755,24.955,154.518
C05162=1069.609,29.170,-65.960,172.754,24.952,154.518
C05163=1069.604,28.920,-65.944,172.753,24.949,154.518
C05164=1069.598,28.670,-65.929,172.751,24.947,154.517
C05165=1069.591,28.421,-65.913,172.750,24.944,154.517
C05166=1069.586,28.172,-65.898,172.749,24.941,154.517
C05167=1069.580,27.922,-65.883,172.747,24.939,154.516
C05168=1069.574,27.673,-65.867,172.746,24.936,154.516
C05169=1069.568,27.423,-65.852,172.745,24.934,154.516
C05170=1069.562,27.174,-65.836,172.743,24.931,154.515
C05171=1069.556,26.925,-65.821,172.742,24.928,154.515
C05172=1069.550,26.675,-65.806,172.741,24.926,154.515
C05173=1069.544,26.425,-65.791,172.739,24.923,154.514
C05174=1069.538,26.176,-65.774,172.738,24.921,154.514
C05175=1069.532,25.927,-65.760,172.737,24.918,154.514
C05176=1069.526,25.677,-65.744,172.735,24.916,154.513
C05177=1069.520,25.428,-65.729,172.734,24.913,154.513
C05178=1069.514,25.178,-65.713,172.732,24.910,154.513
C05179=1069.508,24.929,-65.698,172.731,24.908,154.512
C05180=1069.503,24.679,-65.683,172.730,24.905,154.512
C05181=1069.496,24.430,-65.667,172.728,24.903,154.512
C05182=1069.490,24.180,-65.652,172.726,24.899,154.511
C05183=1069.485,23.931,-65.637,172.725,24.897,154.511
C05184=1069.479,23.681,-65.622,172.724,24.894,154.511
C05185=1069.472,23.432,-65.606,172.722,24.892,154.510
C05186=1069.467,23.183,-65.591,172.721,24.889,154.510
C05187=1069.461,22.933,-65.576,172.719,24.886,154.510
C05188=1069.454,22.684,-65.561,172.718,24.884,154.509
C05189=1069.449,22.434,-65.545,172.717,24.881,154.509
C05190=1069.443,22.185,-65.530,172.715,24.879,154.509
C05191=1069.437,21.935,-65.514,172.714,24.876,154.508
C05192=1069.431,21.686,-65.499,172.713,24.874,154.508
C05193=1069.426,21.436,-65.484,172.711,24.871,154.508
C05194=1069.419,21.187,-65.469,172.710,24.868,154.507
C05195=1069.413,20.937,-65.454,172.709,24.866,154.507
C05196=1069.408,20.688,-65.439,172.707,24.863,154.507
C05197=1069.401,20.439,-65.424,172.706,24.861,154.506
C05198=1069.395,20.189,-65.408,172.705,24.858,154.506
C05199=1069.390,19.940,-65.393,172.703,24.855,154.506
C05200=1069.383,19.690,-65.379,172.702,24.853,154.506
C05201=1069.378,19.440,-65.363,172.701,24.850,154.505
C05202=1069.372,19.191,-65.348,172.699,24.848,154.505
C05203=1069.365,18.942,-65.333,172.698,24.845,154.505
C05204=1069.360,18.692,-65.318,172.697,24.842,154.504
C05205=1069.354,18.443,-65.303,172.695,24.840,154.504
C05206=1069.348,18.193,-65.288,172.694,24.837,154.504
C05207=1069.342,17.943,-65.273,172.692,24.835,154.503
C05208=1069.336,17.694,-65.258,172.691,24.832,154.503
C05209=1069.330,17.444,-65.243,172.689,24.829,154.503
C05210=1069.323,17.195,-65.228,172.687,24.827,154.502
C05211=1069.318,16.946,-65.212,172.686,24.824,154.502
C05212=1069.312,16.697,-65.198,172.685,24.822,154.502
C05213=1069.305,16.447,-65.183,172.683,24.819,154.501
C05214=1069.301,16.197,-65.168,172.682,24.816,154.501
C05215=1069.294,15.947,-65.153,172.681,24.814,154.501
C05216=1069.288,15.698,-65.139,172.679,24.812,154.500
C05217=1069.282,15.449,-65.124,172.678,24.809,154.500
C05218=1069.276,15.199,-65.108,172.677,24.806,154.500
C05219=1069.271,14.950,-65.094,172.675,24.803,154.499
C05220=1069.264,14.668,-65.076,172.674,24.801,154.499
C05221=1069.257,14.387,-65.060,172.673,24.798,154.499
C05222=1069.250,14.105,-65.042,172.671,24.795,154.498
C05223=1069.243,13.824,-65.027,172.669,24.792,154.498
C05224=1069.237,13.575,-65.012,172.668,24.790,154.498
C05225=1069.231,13.326,-64.997,172.666,24.787,154.497
C05226=1069.226,13.076,-64.982,172.665,24.785,154.497
C05227=1069.219,12.826,-64.967,172.664,24.782,154.497
C05228=1069.213,12.577,-64.952,172.662,24.780,154.496
C05229=1069.207,12.327,-64.937,172.661,24.777,154.496
C05230=1069.201,12.077,-64.923,172.660,24.775,154.496
C05231=1069.195,11.828,-64.908,172.658,24.772,154.495
C05232=1069.189,11.578,-64.893,172.657,24.769,154.495
C05233=1069.183,11.330,-64.879,172.656,24.767,154.495
C05234=1069.177,11.080,-64.864,172.653,24.764,154.495
C05235=1069.170,10.830,-64.849,172.652,24.761,154.494
C05236=1069.165,10.581,-64.835,172.651,24.759,154.494
C05237=1069.158,10.331,-64.820,172.649,24.757,154.494
C05238=1069.153,10.082,-64.805,172.648,24.754,154.493
C05239=1069.146,9.832,-64.791,172.647,24.751,154.493
C05240=1069.140,9.583,-64.776,172.645,24.749,154.493
C05241=1069.134,9.333,-64.762,172.644,24.747,154.492
C05242=1069.128,9.084,-64.747,172.642,24.744,154.492
C05243=1069.122,8.835,-64.732,172.641,24.741,154.492
C05244=1069.116,8.585,-64.717,172.640,24.739,154.492
C05245=1069.110,8.335,-64.703,172.638,24.737,154.491
C05246=1069.105,8.085,-64.688,172.637,24.734,154.491
C05247=1069.099,7.836,-64.673,172.636,24.731,154.491
C05248=1069.092,7.587,-64.658,172.634,24.729,154.490
C05249=1069.087,7.337,-64.644,172.633,24.727,154.490
C05250=1069.081,7.087,-64.630,172.632,24.724,154.490
C05251=1069.075,6.839,-64.615,172.630,24.721,154.489
C05252=1069.069,6.588,-64.601,172.629,24.719,154.489
C05253=1069.063,6.339,-64.586,172.627,24.717,154.489
C05254=1069.057,6.090,-64.571,172.626,24.714,154.488
C05255=1069.051,5.840,-64.557,172.625,24.711,154.488
C05256=1069.045,5.590,-64.542,172.623,24.709,154.488
C05257=1069.039,5.341,-64.528,172.622,24.706,154.487
C05258=1069.033,5.091,-64.514,172.621,24.704,154.487
C05259=1069.027,4.842,-64.499,172.619,24.701,154.487
C05260=1069.021,4.593,-64.484,172.618,24.699,154.487
C05261=1069.015,4.343,-64.470,172.616,24.696,154.486
C05262=1069.009,4.093,-64.455,172.614,24.693,154.486
C05263=1069.003,3.844,-64.441,172.613,24.691,154.486
C05264=1068.996,3.594,-64.427,172.612,24.689,154.485
C05265=1068.990,3.345,-64.412,172.610,24.686,154.485
C05266=1068.985,3.096,-64.399,172.609,24.683,154.485
C05267=1068.979,2.846,-64.384,172.607,24.681,154.484
C05268=1068.973,2.597,-64.370,172.606,24.679,154.484
C05269=1068.967,2.347,-64.355,172.605,24.676,154.484
C05270=1068.961,2.098,-64.340,172.603,24.673,154.484
C05271=1068.955,1.848,-64.326,172.602,24.671,154.483
C05272=1068.949,1.599,-64.311,172.601,24.668,154.483
C05273=1068.944,1.349,-64.298,172.599,24.666,154.483
C05274=1068.937,1.100,-64.283,172.598,24.663,154.482
C05275=1068.932,0.850,-64.269,172.597,24.661,154.482
C05276=1068.925,0.600,-64.254,172.595,24.658,154.482
C05277=1068.920,0.351,-64.240,172.594,24.655,154.481
C05278=1068.914,0.102,-64.225,172.593,24.653,154.481
C05279=1068.908,-0.148,-64.211,172.591,24.651,154.481
C05280=1068.902,-0.397,-64.197,172.590,24.648,154.481
C05281=1068.896,-0.648,-64.182,172.589,24.645,154.480
C05282=1068.890,-0.897,-64.168,172.587,24.643,154.480
C05283=1068.885,-1.146,-64.154,172.586,24.641,154.480
C05284=1068.878,-1.426,-64.138,172.584,24.637,154.479
C05285=1068.871,-1.705,-64.122,172.582,24.635,154.479
C05286=1068.865,-1.985,-64.107,172.581,24.632,154.479
C05287=1068.858,-2.264,-64.090,172.579,24.629,154.478
C05288=1068.852,-2.513,-64.076,172.577,24.626,154.478
C05289=1068.846,-2.764,-64.062,172.576,24.624,154.478
C05290=1068.841,-3.012,-64.047,172.575,24.622,154.477
C05291=1068.835,-3.262,-64.033,172.573,24.619,154.477
C05292=1068.828,-3.512,-64.020,172.572,24.616,154.477
C05293=1068.823,-3.761,-64.005,172.571,24.614,154.476
C05294=1068.816,-4.011,-63.991,172.569,24.612,154.476
C05295=1068.810,-4.260,-63.978,172.568,24.609,154.476
C05296=1068.804,-4.509,-63.963,172.566,24.607,154.476
C05297=1068.798,-4.760,-63.949,172.565,24.605,154.475
C05298=1068.792,-5.009,-63.935,172.564,24.602,154.475
C05299=1068.786,-5.259,-63.920,172.562,24.600,154.475
C05300=1068.780,-5.508,-63.907,172.561,24.597,154.475
C05301=1068.774,-5.757,-63.893,172.560,24.594,154.474
C05302=1068.768,-6.007,-63.878,172.558,24.592,154.474
C05303=1068.762,-6.257,-63.865,172.557,24.590,154.474
C05304=1068.756,-6.506,-63.851,172.555,24.587,154.473
C05305=1068.750,-6.756,-63.837,172.554,24.585,154.473
C05306=1068.743,-7.005,-63.823,172.553,24.583,154.473
C05307=1068.738,-7.254,-63.809,172.551,24.580,154.472
C05308=1068.732,-7.505,-63.795,172.550,24.578,154.472
C05309=1068.726,-7.754,-63.782,172.549,24.575,154.472
C05310=1068.720,-8.003,-63.767,172.546,24.573,154.472
C05311=1068.714,-8.253,-63.753,172.545,24.570,154.471
C05312=1068.708,-8.503,-63.740,172.543,24.568,154.471
C05313=1068.702,-8.752,-63.726,172.542,24.566,154.471
C05314=1068.695,-9.001,-63.711,172.541,24.563,154.470
C05315=1068.689,-9.251,-63.698,172.539,24.560,154.470
C05316=1068.684,-9.501,-63.684,172.538,24.558,154.470
C05317=1068.677,-9.751,-63.670,172.537,24.556,154.470
C05318=1068.672,-10.000,-63.656,172.535,24.553,154.469
C05319=1068.665,-10.249,-63.642,172.534,24.551,154.469
C05320=1068.660,-10.498,-63.628,172.533,24.548,154.469
C05321=1068.654,-10.749,-63.614,172.531,24.546,154.469
C05322=1068.647,-10.998,-63.601,172.530,24.544,154.468
C05323=1068.642,-11.247,-63.587,172.528,24.541,154.468
C05324=1068.636,-11.497,-63.574,172.527,24.539,154.468
C05325=1068.630,-11.747,-63.559,172.526,24.536,154.467
C05326=1068.624,-11.997,-63.546,172.524,24.534,154.467
C05327=1068.618,-12.245,-63.532,172.523,24.532,154.467
C05328=1068.612,-12.495,-63.518,172.521,24.529,154.467
C05329=1068.605,-12.745,-63.504,172.520,24.527,154.466
C05330=1068.600,-12.994,-63.490,172.519,24.525,154.466
C05331=1068.594,-13.244,-63.477,172.517,24.522,154.466
C05332=1068.588,-13.493,-63.463,172.516,24.519,154.465
C05333=1068.582,-13.743,-63.449,172.514,24.517,154.465
C05334=1068.576,-13.993,-63.436,172.512,24.514,154.465
C05335=1068.570,-14.242,-63.422,172.511,24.512,154.465
C05336=1068.564,-14.492,-63.408,172.510,24.509,154.464
C05337=1068.559,-14.741,-63.395,172.508,24.507,154.464
C05338=1068.552,-14.991,-63.381,172.507,24.505,154.464
C05339=1068.546,-15.241,-63.367,172.505,24.502,154.464
C05340=1068.540,-15.490,-63.354,172.504,24.500,154.463
C05341=1068.535,-15.740,-63.340,172.503,24.497,154.463
C05342=1068.528,-15.989,-63.326,172.501,24.496,154.463
C05343=1068.522,-16.239,-63.313,172.500,24.493,154.463
C05344=1068.516,-16.488,-63.299,172.498,24.491,154.462
C05345=1068.510,-16.738,-63.286,172.497,24.489,154.462
C05346=1068.503,-16.988,-63.272,172.496,24.486,154.462
C05347=1068.498,-17.237,-63.258,172.494,24.484,154.461
C05348=1068.491,-17.514,-63.244,172.493,24.481,154.461
C05349=1068.484,-17.792,-63.229,172.491,24.478,154.461
C05350=1068.477,-18.070,-63.213,172.489,24.476,154.461
C05351=1068.470,-18.348,-63.199,172.488,24.473,154.460
C05352=1068.465,-18.598,-63.185,172.487,24.471,154.460
C05353=1068.459,-18.847,-63.172,172.485,24.469,154.460
C05354=1068.453,-19.097,-63.157,172.484,24.466,154.459
C05355=1068.446,-19.346,-63.144,172.482,24.463,154.459
C05356=1068.440,-19.596,-63.132,172.480,24.462,154.459
C05357=1068.435,-19.846,-63.118,172.479,24.459,154.459
C05358=1068.429,-20.095,-63.104,172.477,24.457,154.459
C05359=1068.423,-20.344,-63.091,172.476,24.454,154.458
C05360=1068.417,-20.595,-63.077,172.474,24.452,154.458
C05361=1068.410,-20.844,-63.064,172.473,24.450,154.458
C05362=1068.404,-21.093,-63.050,172.472,24.447,154.457
C05363=1068.398,-21.343,-63.038,172.470,24.445,154.457
C05364=1068.393,-21.593,-63.024,172.469,24.443,154.457
C05365=1068.386,-21.842,-63.011,172.467,24.441,154.457
C05366=1068.380,-22.091,-62.997,172.466,24.438,154.457
C05367=1068.374,-22.342,-62.983,172.465,24.436,154.456
C05368=1068.368,-22.591,-62.971,172.463,24.434,154.456
C05369=1068.362,-22.841,-62.957,172.462,24.431,154.456
C05370=1068.357,-23.090,-62.944,172.461,24.429,154.455
C05371=1068.350,-23.339,-62.930,172.459,24.426,154.455
C05372=1068.344,-23.589,-62.918,172.458,24.424,154.455
C05373=1068.338,-23.839,-62.904,172.456,24.422,154.455
C05374=1068.333,-24.088,-62.891,172.455,24.420,154.454
C05375=1068.327,-24.337,-62.877,172.453,24.417,154.454
C05376=1068.321,-24.587,-62.865,172.451,24.415,154.454
C05377=1068.315,-24.838,-62.851,172.450,24.412,154.454
C05378=1068.308,-25.087,-62.837,172.448,24.410,154.453
C05379=1068.302,-25.336,-62.824,172.447,24.407,154.453
C05380=1068.296,-25.586,-62.811,172.446,24.406,154.453
C05381=1068.291,-25.836,-62.798,172.444,24.403,154.453
C05382=1068.285,-26.085,-62.784,172.443,24.401,154.452
C05383=1068.279,-26.335,-62.772,172.441,24.399,154.452
C05384=1068.272,-26.584,-62.758,172.440,24.396,154.452
C05385=1068.267,-26.834,-62.745,172.439,24.394,154.452
C05386=1068.261,-27.083,-62.732,172.437,24.392,154.451
C05387=1068.255,-27.333,-62.719,172.436,24.390,154.451
C05388=1068.249,-27.582,-62.706,172.434,24.387,154.451
C05389=1068.243,-27.832,-62.693,172.433,24.385,154.451
C05390=1068.236,-28.082,-62.679,172.432,24.383,154.451
C05391=1068.230,-28.332,-62.667,172.430,24.381,154.450
C05392=1068.224,-28.581,-62.654,172.429,24.378,154.450
C05393=1068.218,-28.830,-62.640,172.427,24.376,154.450
C05394=1068.212,-29.080,-62.628,172.426,24.374,154.450
C05395=1068.205,-29.329,-62.614,172.424,24.371,154.449
C05396=1068.200,-29.579,-62.602,172.422,24.369,154.449
C05397=1068.193,-29.829,-62.589,172.421,24.367,154.449
C05398=1068.188,-30.079,-62.575,172.419,24.365,154.449
C05399=1068.182,-30.328,-62.562,172.418,24.363,154.448
C05400=1068.176,-30.577,-62.549,172.416,24.360,154.448
C05401=1068.170,-30.827,-62.536,172.415,24.358,154.448
C05402=1068.164,-31.076,-62.523,172.414,24.356,154.448
C05403=1068.158,-31.326,-62.511,172.412,24.354,154.448
C05404=1068.151,-31.576,-62.497,172.411,24.351,154.447
C05405=1068.146,-31.825,-62.485,172.409,24.349,154.447
C05406=1068.139,-32.075,-62.471,172.408,24.347,154.447
C05407=1068.133,-32.325,-62.459,172.407,24.345,154.447
C05408=1068.127,-32.574,-62.446,172.405,24.342,154.446
C05409=1068.121,-32.824,-62.433,172.404,24.341,154.446
C05410=1068.115,-33.074,-62.421,172.402,24.338,154.446
C05411=1068.109,-33.323,-62.407,172.401,24.336,154.446
C05412=1068.102,-33.601,-62.393,172.399,24.333,154.445
C05413=1068.096,-33.877,-62.379,172.397,24.331,154.445
C05414=1068.089,-34.155,-62.364,172.396,24.329,154.445
C05415=1068.082,-34.431,-62.350,172.393,24.326,154.445
C05416=1068.076,-34.681,-62.337,172.392,24.324,154.444
C05417=1068.070,-34.931,-62.325,172.391,24.321,154.444
C05418=1068.064,-35.180,-62.312,172.389,24.319,154.444
C05419=1068.058,-35.430,-62.299,172.388,24.317,154.444
C05420=1068.052,-35.679,-62.286,172.386,24.315,154.444
C05421=1068.046,-35.929,-62.273,172.385,24.313,154.443
C05422=1068.040,-36.179,-62.261,172.384,24.310,154.443
C05423=1068.034,-36.428,-62.247,172.382,24.308,154.443
C05424=1068.029,-36.677,-62.235,172.381,24.306,154.443
C05425=1068.023,-36.927,-62.223,172.379,24.304,154.442
C05426=1068.016,-37.177,-62.209,172.378,24.302,154.442
C05427=1068.011,-37.427,-62.197,172.376,24.300,154.442
C05428=1068.005,-37.676,-62.184,172.375,24.297,154.442
C05429=1067.998,-37.926,-62.171,172.373,24.295,154.442
C05430=1067.993,-38.176,-62.158,172.372,24.293,154.441
C05431=1067.987,-38.425,-62.146,172.371,24.291,154.441
C05432=1067.980,-38.675,-62.133,172.369,24.289,154.441
C05433=1067.974,-38.924,-62.121,172.367,24.286,154.441
C05434=1067.968,-39.174,-62.108,172.365,24.284,154.441
C05435=1067.962,-39.423,-62.095,172.364,24.282,154.440
C05436=1067.956,-39.673,-62.082,172.363,24.280,154.440
C05437=1067.950,-39.922,-62.071,172.361,24.278,154.440
C05438=1067.944,-40.172,-62.058,172.360,24.276,154.440
C05439=1067.938,-40.421,-62.045,172.358,24.274,154.440
C05440=1067.932,-40.671,-62.032,172.357,24.271,154.439
C05441=1067.926,-40.921,-62.020,172.355,24.270,154.439
C05442=1067.919,-41.171,-62.008,172.354,24.267,154.439
C05443=1067.913,-41.421,-61.995,172.352,24.265,154.439
C05444=1067.907,-41.670,-61.982,172.351,24.263,154.438
C05445=1067.901,-41.920,-61.969,172.349,24.261,154.438
C05446=1067.894,-42.169,-61.957,172.348,24.259,154.438
C05447=1067.889,-42.419,-61.945,172.347,24.257,154.438
C05448=1067.883,-42.668,-61.933,172.345,24.255,154.438
C05449=1067.877,-42.918,-61.919,172.344,24.253,154.437
C05450=1067.870,-43.167,-61.907,172.342,24.251,154.437
C05451=1067.864,-43.417,-61.895,172.340,24.248,154.437
C05452=1067.859,-43.667,-61.882,172.338,24.246,154.437
C05453=1067.852,-43.916,-61.870,172.337,24.244,154.437
C05454=1067.846,-44.166,-61.858,172.336,24.242,154.437
